LIN {X -0.292,Y -605.809,Z 406.567,A 0.000,B 0.000,C 90.000,E1 318.081} C_DIS
LIN {X 0.319,Y -611.269,Z 406.558,A 0.000,B 0.000,C 90.000,E1 316.458} C_DIS
LIN {X 0.160,Y -616.740,Z 406.550,A 0.000,B 0.000,C 90.000,E1 314.919} C_DIS
LIN {X -0.037,Y -623.235,Z 406.540,A 0.000,B 0.000,C 90.000,E1 313.137} C_DIS
LIN {X -0.138,Y -626.967,Z 406.534,A 0.000,B 0.000,C 90.000,E1 312.123} C_DIS
LIN {X -0.379,Y -632.521,Z 406.526,A 0.000,B 0.000,C 90.000,E1 310.620} C_DIS
LIN {X 0.008,Y -636.977,Z 406.518,A 0.000,B 0.000,C 90.000,E1 309.322} C_DIS
LIN {X 0.062,Y -641.986,Z 406.510,A 0.000,B 0.000,C 90.000,E1 307.810} C_DIS
LIN {X -0.197,Y -646.015,Z 406.503,A 0.000,B 0.000,C 90.000,E1 306.583} C_DIS
LIN {X 0.128,Y -649.848,Z 406.496,A 0.000,B 0.000,C 90.000,E1 305.311} C_DIS
LIN {X 0.149,Y -653.624,Z 406.489,A 0.000,B 0.000,C 90.000,E1 304.072} C_DIS
LIN {X -0.214,Y -657.959,Z 406.481,A 0.000,B 0.000,C 90.000,E1 302.625} C_DIS
LIN {X 0.054,Y -662.210,Z 406.473,A 0.000,B 0.000,C 90.000,E1 301.131} C_DIS
LIN {X 0.058,Y -666.331,Z 406.465,A 0.000,B 0.000,C 90.000,E1 299.667} C_DIS
LIN {X -0.349,Y -669.415,Z 406.458,A 0.000,B 0.000,C 90.000,E1 298.487} C_DIS
LIN {X 0.140,Y -671.219,Z 406.454,A 0.000,B 0.000,C 90.000,E1 297.719} C_DIS
LIN {X -0.141,Y -674.920,Z 406.445,A 0.000,B 0.000,C 90.000,E1 296.052} C_DIS
LIN {X -0.017,Y -676.898,Z 406.439,A 0.000,B 0.000,C 90.000,E1 295.079} C_DIS
LIN {X -0.164,Y -678.756,Z 406.434,A 0.000,B 0.000,C 90.000,E1 294.131} C_DIS
LIN {X 0.259,Y -680.450,Z 406.427,A 0.000,B 0.000,C 90.000,E1 292.898} C_DIS
LIN {X -0.046,Y -681.185,Z 406.423,A 0.000,B 0.000,C 90.000,E1 292.206} C_DIS
LIN {X 0.227,Y -681.792,Z 406.418,A 0.000,B 0.000,C 90.000,E1 291.227} C_DIS
LIN {X -0.127,Y -682.278,Z 406.413,A 0.000,B 0.000,C 90.000,E1 290.301} C_DIS
LIN {X -0.027,Y -682.414,Z 406.409,A 0.000,B 0.000,C 90.000,E1 289.577} C_DIS
LIN {X 0.259,Y -682.311,Z 406.404,A 0.000,B 0.000,C 90.000,E1 288.598} C_DIS
LIN {X 0.359,Y -681.967,Z 406.400,A 0.000,B 0.000,C 90.000,E1 287.873} C_DIS
LIN {X -0.234,Y -681.446,Z 406.394,A 0.000,B 0.000,C 90.000,E1 286.968} C_DIS
LIN {X 0.245,Y -680.502,Z 406.388,A 0.000,B 0.000,C 90.000,E1 285.733} C_DIS
LIN {X 0.357,Y -680.103,Z 406.385,A 0.000,B 0.000,C 90.000,E1 285.245} C_DIS
LIN {X 0.127,Y -678.512,Z 406.377,A 0.000,B 0.000,C 90.000,E1 283.828} C_DIS
LIN {X -0.041,Y -677.497,Z 406.372,A 0.000,B 0.000,C 90.000,E1 282.883} C_DIS
LIN {X -0.370,Y -676.465,Z 406.366,A 0.000,B 0.000,C 90.000,E1 281.951} C_DIS
LIN {X 0.335,Y -673.842,Z 406.354,A 0.000,B 0.000,C 90.000,E1 279.726} C_DIS
LIN {X -0.044,Y -671.489,Z 406.342,A 0.000,B 0.000,C 90.000,E1 277.587} C_DIS
LIN {X 0.176,Y -669.413,Z 406.330,A 0.000,B 0.000,C 90.000,E1 275.391} C_DIS
LIN {X -0.191,Y -667.809,Z 406.321,A 0.000,B 0.000,C 90.000,E1 273.726} C_DIS
LIN {X 0.028,Y -667.186,Z 406.317,A 0.000,B 0.000,C 90.000,E1 272.980} C_DIS
LIN {X 0.079,Y -665.517,Z 406.306,A 0.000,B 0.000,C 90.000,E1 271.031} C_DIS
LIN {X -0.082,Y -664.332,Z 406.299,A 0.000,B 0.000,C 90.000,E1 269.828} C_DIS
LIN {X 0.247,Y -663.720,Z 406.296,A 0.000,B 0.000,C 90.000,E1 269.312} C_DIS
LIN {X 0.078,Y -663.348,Z 406.295,A 0.000,B 0.000,C 90.000,E1 269.083} C_DIS
LIN {X -0.092,Y -663.132,Z 406.294,A 0.000,B 0.000,C 90.000,E1 268.854} C_DIS
LIN {X -0.278,Y -661.542,Z 406.287,A 0.000,B 0.000,C 90.000,E1 267.650} C_DIS
LIN {X 0.175,Y -659.739,Z 406.280,A 0.000,B 0.000,C 90.000,E1 266.388} C_DIS
LIN {X 0.316,Y -658.453,Z 406.276,A 0.000,B 0.000,C 90.000,E1 265.641} C_DIS
LIN {X -0.212,Y -656.934,Z 406.272,A 0.000,B 0.000,C 90.000,E1 264.951} C_DIS
LIN {X -0.239,Y -654.722,Z 406.266,A 0.000,B 0.000,C 90.000,E1 263.970} C_DIS
LIN {X 0.134,Y -651.558,Z 406.260,A 0.000,B 0.000,C 90.000,E1 262.704} C_DIS
LIN {X -0.260,Y -647.578,Z 406.251,A 0.000,B 0.000,C 90.000,E1 261.254} C_DIS
LIN {X 0.061,Y -643.908,Z 406.244,A 0.000,B 0.000,C 90.000,E1 259.982} C_DIS
LIN {X 0.256,Y -639.424,Z 406.236,A 0.000,B 0.000,C 90.000,E1 258.465} C_DIS
LIN {X -0.125,Y -634.791,Z 406.228,A 0.000,B 0.000,C 90.000,E1 256.992} C_DIS
LIN {X -0.219,Y -631.533,Z 406.222,A 0.000,B 0.000,C 90.000,E1 255.992} C_DIS
LIN {X 0.247,Y -628.136,Z 406.216,A 0.000,B 0.000,C 90.000,E1 254.936} C_DIS
LIN {X 0.009,Y -623.629,Z 406.209,A 0.000,B 0.000,C 90.000,E1 253.685} C_DIS
LIN {X -0.080,Y -619.921,Z 406.204,A 0.000,B 0.000,C 90.000,E1 252.670} C_DIS
LIN {X -0.030,Y -616.128,Z 406.198,A 0.000,B 0.000,C 90.000,E1 251.638} C_DIS
LIN {X -0.277,Y -611.249,Z 406.191,A 0.000,B 0.000,C 90.000,E1 250.369} C_DIS
LIN {X 0.167,Y -606.185,Z 406.184,A 0.000,B 0.000,C 90.000,E1 249.028} C_DIS
LIN {X 0.177,Y -600.901,Z 406.176,A 0.000,B 0.000,C 90.000,E1 247.720} C_DIS
LIN {X 0.192,Y -596.560,Z 406.171,A 0.000,B 0.000,C 90.000,E1 246.666} C_DIS
LIN {X -0.057,Y -589.938,Z 406.162,A 0.000,B 0.000,C 90.000,E1 245.101} C_DIS
LIN {X -0.316,Y -582.091,Z 406.151,A 0.000,B 0.000,C 90.000,E1 243.256} C_DIS
LIN {X -0.206,Y -576.508,Z 406.144,A 0.000,B 0.000,C 90.000,E1 241.897} C_DIS
LIN {X -0.254,Y -568.849,Z 406.133,A 0.000,B 0.000,C 90.000,E1 239.999} C_DIS
LIN {X -0.120,Y -560.426,Z 406.121,A 0.000,B 0.000,C 90.000,E1 237.788} C_DIS
LIN {X 0.063,Y -552.448,Z 406.109,A 0.000,B 0.000,C 90.000,E1 235.548} C_DIS
LIN {X 0.040,Y -547.623,Z 406.101,A 0.000,B 0.000,C 90.000,E1 234.149} C_DIS
LIN {X -0.181,Y -542.844,Z 406.093,A 0.000,B 0.000,C 90.000,E1 232.763} C_DIS
LIN {X -0.052,Y -538.005,Z 406.085,A 0.000,B 0.000,C 90.000,E1 231.331} C_DIS
LIN {X -0.102,Y -532.284,Z 406.076,A 0.000,B 0.000,C 90.000,E1 229.622} C_DIS
LIN {X -0.047,Y -525.042,Z 406.063,A 0.000,B 0.000,C 90.000,E1 227.310} C_DIS
LIN {X -0.064,Y -519.755,Z 406.053,A 0.000,B 0.000,C 90.000,E1 225.567} C_DIS
LIN {X 0.164,Y -514.572,Z 406.043,A 0.000,B 0.000,C 90.000,E1 223.785} C_DIS
LIN {X -0.087,Y -509.453,Z 406.034,A 0.000,B 0.000,C 90.000,E1 222.043} C_DIS
LIN {X 0.189,Y -503.698,Z 406.022,A 0.000,B 0.000,C 90.000,E1 219.930} C_DIS
LIN {X -0.009,Y -498.183,Z 406.010,A 0.000,B 0.000,C 90.000,E1 217.855} C_DIS
LIN {X -0.273,Y -494.353,Z 406.002,A 0.000,B 0.000,C 90.000,E1 216.377} C_DIS
LIN {X 0.179,Y -489.131,Z 405.990,A 0.000,B 0.000,C 90.000,E1 214.199} C_DIS
LIN {X 0.154,Y -485.555,Z 405.982,A 0.000,B 0.000,C 90.000,E1 212.673} C_DIS
LIN {X 0.011,Y -481.312,Z 405.971,A 0.000,B 0.000,C 90.000,E1 210.846} C_DIS
LIN {X -0.097,Y -476.330,Z 405.959,A 0.000,B 0.000,C 90.000,E1 208.693} C_DIS
LIN {X 0.003,Y -473.428,Z 405.952,A 0.000,B 0.000,C 90.000,E1 207.436} C_DIS
LIN {X 0.045,Y -470.495,Z 405.946,A 0.000,B 0.000,C 90.000,E1 206.181} C_DIS
LIN {X -0.225,Y -466.721,Z 405.937,A 0.000,B 0.000,C 90.000,E1 204.643} C_DIS
LIN {X 0.150,Y -463.676,Z 405.930,A 0.000,B 0.000,C 90.000,E1 203.334} C_DIS
LIN {X 0.237,Y -458.340,Z 405.917,A 0.000,B 0.000,C 90.000,E1 201.099} C_DIS
LIN {X 0.173,Y -452.612,Z 405.903,A 0.000,B 0.000,C 90.000,E1 198.544} C_DIS
LIN {X -0.081,Y -448.051,Z 405.891,A 0.000,B 0.000,C 90.000,E1 196.315} C_DIS
LIN {X -0.004,Y -443.326,Z 405.876,A 0.000,B 0.000,C 90.000,E1 193.703} C_DIS
LIN {X 0.182,Y -440.022,Z 405.865,A 0.000,B 0.000,C 90.000,E1 191.715} C_DIS
LIN {X -0.225,Y -435.417,Z 405.849,A 0.000,B 0.000,C 90.000,E1 188.803} C_DIS
LIN {X 0.182,Y -432.241,Z 405.836,A 0.000,B 0.000,C 90.000,E1 186.429} C_DIS
LIN {X -0.068,Y -429.477,Z 405.823,A 0.000,B 0.000,C 90.000,E1 184.131} C_DIS
LIN {X -0.109,Y -427.760,Z 405.814,A 0.000,B 0.000,C 90.000,E1 182.465} C_DIS
LIN {X 0.028,Y -425.302,Z 405.797,A 0.000,B 0.000,C 90.000,E1 179.427} C_DIS
LIN {X -0.092,Y -423.384,Z 405.773,A 0.000,B 0.000,C 90.000,E1 175.065} C_DIS
LIN {X -0.099,Y -423.234,Z 405.748,A 0.000,B 0.000,C 90.000,E1 170.679} C_DIS
LIN {X -0.112,Y -424.257,Z 405.731,A 0.000,B 0.000,C 90.000,E1 167.645} C_DIS
LIN {X 0.010,Y -425.939,Z 405.716,A 0.000,B 0.000,C 90.000,E1 164.936} C_DIS
LIN {X -0.203,Y -429.303,Z 405.696,A 0.000,B 0.000,C 90.000,E1 161.275} C_DIS
LIN {X 0.081,Y -432.036,Z 405.683,A 0.000,B 0.000,C 90.000,E1 158.901} C_DIS
LIN {X -0.211,Y -435.267,Z 405.670,A 0.000,B 0.000,C 90.000,E1 156.613} C_DIS
LIN {X 0.056,Y -441.290,Z 405.650,A 0.000,B 0.000,C 90.000,E1 152.948} C_DIS
LIN {X 0.241,Y -448.469,Z 405.630,A 0.000,B 0.000,C 90.000,E1 149.331} C_DIS
LIN {X -0.188,Y -453.751,Z 405.617,A 0.000,B 0.000,C 90.000,E1 147.120} C_DIS
LIN {X 0.011,Y -459.606,Z 405.605,A 0.000,B 0.000,C 90.000,E1 144.848} C_DIS
LIN {X 0.058,Y -467.981,Z 405.589,A 0.000,B 0.000,C 90.000,E1 141.984} C_DIS
LIN {X 0.168,Y -475.901,Z 405.575,A 0.000,B 0.000,C 90.000,E1 139.461} C_DIS
LIN {X -0.049,Y -479.829,Z 405.568,A 0.000,B 0.000,C 90.000,E1 138.243} C_DIS
LIN {X 0.117,Y -483.696,Z 405.561,A 0.000,B 0.000,C 90.000,E1 136.986} C_DIS
LIN {X 0.005,Y -487.291,Z 405.554,A 0.000,B 0.000,C 90.000,E1 135.769} C_DIS
LIN {X 0.117,Y -489.885,Z 405.549,A 0.000,B 0.000,C 90.000,E1 134.838} C_DIS
LIN {X 0.084,Y -492.873,Z 405.542,A 0.000,B 0.000,C 90.000,E1 133.623} C_DIS
LIN {X 0.271,Y -495.021,Z 405.537,A 0.000,B 0.000,C 90.000,E1 132.690} C_DIS
LIN {X -0.068,Y -496.262,Z 405.534,A 0.000,B 0.000,C 90.000,E1 132.123} C_DIS
LIN {X -0.032,Y -497.437,Z 405.531,A 0.000,B 0.000,C 90.000,E1 131.515} C_DIS
LIN {X -0.123,Y -498.910,Z 405.526,A 0.000,B 0.000,C 90.000,E1 130.620} C_DIS
LIN {X -0.003,Y -500.317,Z 405.519,A 0.000,B 0.000,C 90.000,E1 129.402} C_DIS
LIN {X -0.064,Y -500.918,Z 405.514,A 0.000,B 0.000,C 90.000,E1 128.508} C_DIS
LIN {X -0.032,Y -500.915,Z 405.509,A 0.000,B 0.000,C 90.000,E1 127.604} C_DIS
LIN {X 0.031,Y -500.539,Z 405.506,A 0.000,B 0.000,C 90.000,E1 126.996} C_DIS
LIN {X 0.068,Y -499.639,Z 405.501,A 0.000,B 0.000,C 90.000,E1 126.091} C_DIS
LIN {X -0.180,Y -498.858,Z 405.497,A 0.000,B 0.000,C 90.000,E1 125.518} C_DIS
LIN {X -0.156,Y -497.379,Z 405.492,A 0.000,B 0.000,C 90.000,E1 124.612} C_DIS
LIN {X 0.122,Y -496.834,Z 405.491,A 0.000,B 0.000,C 90.000,E1 124.278} C_DIS
LIN {X -0.021,Y -493.960,Z 405.484,A 0.000,B 0.000,C 90.000,E1 123.086} C_DIS
LIN {X 0.095,Y -492.235,Z 405.480,A 0.000,B 0.000,C 90.000,E1 122.467} C_DIS
LIN {X -0.064,Y -490.351,Z 405.477,A 0.000,B 0.000,C 90.000,E1 121.878} C_DIS
LIN {X 0.268,Y -487.154,Z 405.472,A 0.000,B 0.000,C 90.000,E1 120.924} C_DIS
LIN {X -0.159,Y -486.075,Z 405.470,A 0.000,B 0.000,C 90.000,E1 120.669} C_DIS
LIN {X -0.123,Y -482.428,Z 405.465,A 0.000,B 0.000,C 90.000,E1 119.745} C_DIS
LIN {X 0.064,Y -477.213,Z 405.458,A 0.000,B 0.000,C 90.000,E1 118.487} C_DIS
LIN {X -0.017,Y -473.070,Z 405.453,A 0.000,B 0.000,C 90.000,E1 117.564} C_DIS
LIN {X -0.180,Y -467.971,Z 405.447,A 0.000,B 0.000,C 90.000,E1 116.488} C_DIS
LIN {X 0.066,Y -459.764,Z 405.437,A 0.000,B 0.000,C 90.000,E1 114.719} C_DIS
LIN {X -0.135,Y -450.626,Z 405.427,A 0.000,B 0.000,C 90.000,E1 112.823} C_DIS
LIN {X -0.023,Y -449.846,Z 405.426,A 0.000,B 0.000,C 90.000,E1 112.642} C_DIS
LIN {X -0.063,Y -449.857,Z 405.426,A 0.000,B 0.000,C 90.000,E1 112.642} C_DIS
LIN {X 0.142,Y -456.999,Z 405.411,A 0.000,B 0.000,C 90.000,E1 109.885} C_DIS
LIN {X -0.050,Y -458.255,Z 405.407,A 0.000,B 0.000,C 90.000,E1 109.268} C_DIS
LIN {X 0.148,Y -466.417,Z 405.386,A 0.000,B 0.000,C 90.000,E1 105.426} C_DIS
LIN {X -0.129,Y -467.925,Z 405.382,A 0.000,B 0.000,C 90.000,E1 104.828} C_DIS
LIN {X -0.015,Y -475.501,Z 405.358,A 0.000,B 0.000,C 90.000,E1 100.423} C_DIS
LIN {X -0.263,Y -476.141,Z 405.356,A 0.000,B 0.000,C 90.000,E1 100.141} C_DIS
LIN {X 0.020,Y -482.054,Z 405.330,A 0.000,B 0.000,C 90.000,E1 95.454} C_DIS
LIN {X -0.190,Y -485.484,Z 405.305,A 0.000,B 0.000,C 90.000,E1 90.859} C_DIS
LIN {X -0.157,Y -486.386,Z 405.281,A 0.000,B 0.000,C 90.000,E1 86.560} C_DIS
LIN {X 0.153,Y -486.363,Z 405.279,A 0.000,B 0.000,C 90.000,E1 86.216} C_DIS
LIN {X 0.236,Y -484.689,Z 405.254,A 0.000,B 0.000,C 90.000,E1 81.602} C_DIS
LIN {X -0.016,Y -483.031,Z 405.245,A 0.000,B 0.000,C 90.000,E1 80.095} C_DIS
LIN {X 0.135,Y -480.621,Z 405.228,A 0.000,B 0.000,C 90.000,E1 76.992} C_DIS
LIN {X -0.007,Y -480.289,Z 405.226,A 0.000,B 0.000,C 90.000,E1 76.700} C_DIS
LIN {X -0.103,Y -474.111,Z 405.200,A 0.000,B 0.000,C 90.000,E1 72.054} C_DIS
LIN {X -0.058,Y -469.651,Z 405.187,A 0.000,B 0.000,C 90.000,E1 69.699} C_DIS
LIN {X -0.099,Y -469.650,Z 405.187,A 0.000,B 0.000,C 90.000,E1 69.699} C_DIS
LIN {X -0.162,Y -479.044,Z 405.180,A 0.000,B 0.000,C 90.000,E1 68.465} C_DIS
LIN {X 0.046,Y -487.179,Z 405.174,A 0.000,B 0.000,C 90.000,E1 67.358} C_DIS
LIN {X 0.117,Y -494.115,Z 405.169,A 0.000,B 0.000,C 90.000,E1 66.433} C_DIS
LIN {X 0.013,Y -500.651,Z 405.164,A 0.000,B 0.000,C 90.000,E1 65.537} C_DIS
LIN {X -0.038,Y -505.900,Z 405.160,A 0.000,B 0.000,C 90.000,E1 64.793} C_DIS
LIN {X -0.007,Y -511.657,Z 405.155,A 0.000,B 0.000,C 90.000,E1 63.896} C_DIS
LIN {X 0.262,Y -516.102,Z 405.151,A 0.000,B 0.000,C 90.000,E1 63.127} C_DIS
LIN {X 0.116,Y -520.139,Z 405.147,A 0.000,B 0.000,C 90.000,E1 62.410} C_DIS
LIN {X 0.083,Y -522.373,Z 405.144,A 0.000,B 0.000,C 90.000,E1 61.975} C_DIS
LIN {X -0.010,Y -525.740,Z 405.140,A 0.000,B 0.000,C 90.000,E1 61.257} C_DIS
LIN {X -0.075,Y -528.710,Z 405.136,A 0.000,B 0.000,C 90.000,E1 60.539} C_DIS
LIN {X -0.005,Y -531.910,Z 405.132,A 0.000,B 0.000,C 90.000,E1 59.665} C_DIS
LIN {X -0.305,Y -532.888,Z 405.130,A 0.000,B 0.000,C 90.000,E1 59.410} C_DIS
LIN {X -0.186,Y -535.279,Z 405.125,A 0.000,B 0.000,C 90.000,E1 58.535} C_DIS
LIN {X -0.033,Y -536.723,Z 405.122,A 0.000,B 0.000,C 90.000,E1 57.946} C_DIS
LIN {X -0.035,Y -538.263,Z 405.117,A 0.000,B 0.000,C 90.000,E1 57.089} C_DIS
LIN {X 0.136,Y -539.104,Z 405.114,A 0.000,B 0.000,C 90.000,E1 56.501} C_DIS
LIN {X -0.128,Y -539.955,Z 405.109,A 0.000,B 0.000,C 90.000,E1 55.674} C_DIS
LIN {X -0.075,Y -540.394,Z 405.105,A 0.000,B 0.000,C 90.000,E1 54.815} C_DIS
LIN {X -0.328,Y -540.511,Z 405.100,A 0.000,B 0.000,C 90.000,E1 53.989} C_DIS
LIN {X -0.265,Y -540.225,Z 405.095,A 0.000,B 0.000,C 90.000,E1 53.130} C_DIS
LIN {X -0.204,Y -539.735,Z 405.090,A 0.000,B 0.000,C 90.000,E1 52.271} C_DIS
LIN {X 0.199,Y -538.721,Z 405.084,A 0.000,B 0.000,C 90.000,E1 51.090} C_DIS
LIN {X -0.178,Y -537.800,Z 405.079,A 0.000,B 0.000,C 90.000,E1 50.275} C_DIS
LIN {X 0.192,Y -536.392,Z 405.073,A 0.000,B 0.000,C 90.000,E1 49.094} C_DIS
LIN {X 0.071,Y -533.908,Z 405.063,A 0.000,B 0.000,C 90.000,E1 47.391} C_DIS
LIN {X -0.151,Y -530.898,Z 405.052,A 0.000,B 0.000,C 90.000,E1 45.405} C_DIS
LIN {X -0.021,Y -528.478,Z 405.043,A 0.000,B 0.000,C 90.000,E1 43.662} C_DIS
LIN {X 0.094,Y -526.657,Z 405.035,A 0.000,B 0.000,C 90.000,E1 42.204} C_DIS
LIN {X 0.159,Y -524.464,Z 405.025,A 0.000,B 0.000,C 90.000,E1 40.458} C_DIS
LIN {X -0.118,Y -522.730,Z 405.017,A 0.000,B 0.000,C 90.000,E1 39.036} C_DIS
LIN {X -0.024,Y -520.969,Z 405.009,A 0.000,B 0.000,C 90.000,E1 37.569} C_DIS
LIN {X 0.083,Y -518.720,Z 404.999,A 0.000,B 0.000,C 90.000,E1 35.804} C_DIS
LIN {X 0.207,Y -516.855,Z 404.991,A 0.000,B 0.000,C 90.000,E1 34.326} C_DIS
LIN {X -0.074,Y -514.486,Z 404.981,A 0.000,B 0.000,C 90.000,E1 32.594} C_DIS
LIN {X 0.183,Y -512.099,Z 404.971,A 0.000,B 0.000,C 90.000,E1 30.797} C_DIS
LIN {X 0.030,Y -509.398,Z 404.960,A 0.000,B 0.000,C 90.000,E1 28.743} C_DIS
LIN {X 0.091,Y -506.540,Z 404.947,A 0.000,B 0.000,C 90.000,E1 26.360} C_DIS
LIN {X 0.217,Y -504.245,Z 404.935,A 0.000,B 0.000,C 90.000,E1 24.259} C_DIS
LIN {X -0.054,Y -501.964,Z 404.922,A 0.000,B 0.000,C 90.000,E1 21.897} C_DIS
LIN {X -0.209,Y -499.869,Z 404.907,A 0.000,B 0.000,C 90.000,E1 19.214} C_DIS
LIN {X -0.141,Y -498.656,Z 404.897,A 0.000,B 0.000,C 90.000,E1 17.402} C_DIS
LIN {X -0.251,Y -497.468,Z 404.887,A 0.000,B 0.000,C 90.000,E1 15.607} C_DIS
LIN {X -0.014,Y -496.319,Z 404.875,A 0.000,B 0.000,C 90.000,E1 13.467} C_DIS
LIN {X 0.073,Y -495.186,Z 404.858,A 0.000,B 0.000,C 90.000,E1 10.433} C_DIS
LIN {X -0.120,Y -494.821,Z 404.840,A 0.000,B 0.000,C 90.000,E1 7.125} C_DIS
LIN {X 0.234,Y -495.290,Z 404.824,A 0.000,B 0.000,C 90.000,E1 4.359} C_DIS
LIN {X 0.114,Y -497.276,Z 404.804,A 0.000,B 0.000,C 90.000,E1 0.745} C_DIS
LIN {X 0.050,Y -500.917,Z 404.784,A 0.000,B 0.000,C 90.000,E1 357.078} C_DIS
LIN {X 0.097,Y -504.640,Z 404.769,A 0.000,B 0.000,C 90.000,E1 354.375} C_DIS
LIN {X 0.231,Y -510.046,Z 404.751,A 0.000,B 0.000,C 90.000,E1 351.084} C_DIS
LIN {X -0.206,Y -517.264,Z 404.731,A 0.000,B 0.000,C 90.000,E1 347.589} C_DIS
LIN {X -0.020,Y -523.695,Z 404.716,A 0.000,B 0.000,C 90.000,E1 344.936} C_DIS
LIN {X 0.138,Y -529.654,Z 404.703,A 0.000,B 0.000,C 90.000,E1 342.598} C_DIS
LIN {X -0.256,Y -534.266,Z 404.694,A 0.000,B 0.000,C 90.000,E1 340.913} C_DIS
LIN {X -0.166,Y -539.823,Z 404.683,A 0.000,B 0.000,C 90.000,E1 338.901} C_DIS
LIN {X 0.015,Y -544.710,Z 404.673,A 0.000,B 0.000,C 90.000,E1 337.177} C_DIS
LIN {X 0.012,Y -549.662,Z 404.664,A 0.000,B 0.000,C 90.000,E1 335.485} C_DIS
LIN {X -0.146,Y -554.736,Z 404.655,A 0.000,B 0.000,C 90.000,E1 333.819} C_DIS
LIN {X 0.099,Y -560.909,Z 404.644,A 0.000,B 0.000,C 90.000,E1 331.847} C_DIS
LIN {X 0.056,Y -564.471,Z 404.638,A 0.000,B 0.000,C 90.000,E1 330.745} C_DIS
LIN {X -0.335,Y -569.001,Z 404.630,A 0.000,B 0.000,C 90.000,E1 329.410} C_DIS
LIN {X 0.142,Y -573.488,Z 404.622,A 0.000,B 0.000,C 90.000,E1 327.995} C_DIS
LIN {X 0.053,Y -578.802,Z 404.613,A 0.000,B 0.000,C 90.000,E1 326.373} C_DIS
LIN {X 0.088,Y -585.073,Z 404.603,A 0.000,B 0.000,C 90.000,E1 324.482} C_DIS
LIN {X -0.199,Y -591.451,Z 404.592,A 0.000,B 0.000,C 90.000,E1 322.637} C_DIS
LIN {X -0.219,Y -598.891,Z 404.581,A 0.000,B 0.000,C 90.000,E1 320.517} C_DIS
LIN {X -0.190,Y -602.702,Z 404.575,A 0.000,B 0.000,C 90.000,E1 319.461} C_DIS
LIN {X -0.307,Y -607.397,Z 404.567,A 0.000,B 0.000,C 90.000,E1 318.162} C_DIS
LIN {X 0.068,Y -611.968,Z 404.560,A 0.000,B 0.000,C 90.000,E1 316.824} C_DIS
LIN {X -0.343,Y -616.514,Z 404.553,A 0.000,B 0.000,C 90.000,E1 315.567} C_DIS
LIN {X 0.192,Y -623.936,Z 404.542,A 0.000,B 0.000,C 90.000,E1 313.461} C_DIS
LIN {X 0.312,Y -629.479,Z 404.533,A 0.000,B 0.000,C 90.000,E1 311.919} C_DIS
LIN {X -0.233,Y -634.141,Z 404.526,A 0.000,B 0.000,C 90.000,E1 310.701} C_DIS
LIN {X 0.185,Y -638.585,Z 404.519,A 0.000,B 0.000,C 90.000,E1 309.402} C_DIS
LIN {X -0.134,Y -642.816,Z 404.512,A 0.000,B 0.000,C 90.000,E1 308.177} C_DIS
LIN {X 0.011,Y -646.880,Z 404.505,A 0.000,B 0.000,C 90.000,E1 306.916} C_DIS
LIN {X -0.126,Y -651.561,Z 404.497,A 0.000,B 0.000,C 90.000,E1 305.438} C_DIS
LIN {X 0.371,Y -655.990,Z 404.489,A 0.000,B 0.000,C 90.000,E1 303.913} C_DIS
LIN {X 0.026,Y -658.914,Z 404.483,A 0.000,B 0.000,C 90.000,E1 302.959} C_DIS
LIN {X -0.281,Y -661.770,Z 404.478,A 0.000,B 0.000,C 90.000,E1 302.005} C_DIS
LIN {X -0.286,Y -665.988,Z 404.470,A 0.000,B 0.000,C 90.000,E1 300.541} C_DIS
LIN {X 0.063,Y -668.735,Z 404.464,A 0.000,B 0.000,C 90.000,E1 299.539} C_DIS
LIN {X 0.119,Y -671.176,Z 404.459,A 0.000,B 0.000,C 90.000,E1 298.565} C_DIS
LIN {X 0.209,Y -673.459,Z 404.453,A 0.000,B 0.000,C 90.000,E1 297.590} C_DIS
LIN {X 0.090,Y -676.595,Z 404.445,A 0.000,B 0.000,C 90.000,E1 296.155} C_DIS
LIN {X -0.252,Y -678.133,Z 404.441,A 0.000,B 0.000,C 90.000,E1 295.463} C_DIS
LIN {X 0.238,Y -679.925,Z 404.436,A 0.000,B 0.000,C 90.000,E1 294.463} C_DIS
LIN {X 0.132,Y -681.298,Z 404.431,A 0.000,B 0.000,C 90.000,E1 293.515} C_DIS
LIN {X -0.164,Y -682.122,Z 404.427,A 0.000,B 0.000,C 90.000,E1 292.823} C_DIS
LIN {X -0.027,Y -682.523,Z 404.424,A 0.000,B 0.000,C 90.000,E1 292.333} C_DIS
LIN {X 0.316,Y -682.912,Z 404.420,A 0.000,B 0.000,C 90.000,E1 291.589} C_DIS
LIN {X -0.072,Y -683.284,Z 404.414,A 0.000,B 0.000,C 90.000,E1 290.429} C_DIS
LIN {X 0.080,Y -683.327,Z 404.411,A 0.000,B 0.000,C 90.000,E1 289.939} C_DIS
LIN {X 0.341,Y -683.100,Z 404.404,A 0.000,B 0.000,C 90.000,E1 288.725} C_DIS
LIN {X -0.232,Y -682.613,Z 404.399,A 0.000,B 0.000,C 90.000,E1 287.819} C_DIS
LIN {X -0.128,Y -682.226,Z 404.395,A 0.000,B 0.000,C 90.000,E1 287.094} C_DIS
LIN {X -0.102,Y -681.144,Z 404.388,A 0.000,B 0.000,C 90.000,E1 285.898} C_DIS
LIN {X -0.171,Y -680.632,Z 404.386,A 0.000,B 0.000,C 90.000,E1 285.426} C_DIS
LIN {X -0.385,Y -678.739,Z 404.378,A 0.000,B 0.000,C 90.000,E1 284.008} C_DIS
LIN {X 0.113,Y -677.597,Z 404.372,A 0.000,B 0.000,C 90.000,E1 283.008} C_DIS
LIN {X -0.069,Y -676.406,Z 404.367,A 0.000,B 0.000,C 90.000,E1 282.063} C_DIS
LIN {X -0.156,Y -673.613,Z 404.355,A 0.000,B 0.000,C 90.000,E1 279.905} C_DIS
LIN {X 0.058,Y -670.894,Z 404.342,A 0.000,B 0.000,C 90.000,E1 277.473} C_DIS
LIN {X -0.299,Y -669.073,Z 404.331,A 0.000,B 0.000,C 90.000,E1 275.568} C_DIS
LIN {X 0.170,Y -667.833,Z 404.323,A 0.000,B 0.000,C 90.000,E1 274.073} C_DIS
LIN {X 0.283,Y -666.289,Z 404.312,A 0.000,B 0.000,C 90.000,E1 272.121} C_DIS
LIN {X 0.152,Y -665.532,Z 404.305,A 0.000,B 0.000,C 90.000,E1 270.917} C_DIS
LIN {X -0.009,Y -664.468,Z 404.298,A 0.000,B 0.000,C 90.000,E1 269.714} C_DIS
LIN {X -0.188,Y -663.195,Z 404.292,A 0.000,B 0.000,C 90.000,E1 268.511} C_DIS
LIN {X -0.022,Y -662.406,Z 404.288,A 0.000,B 0.000,C 90.000,E1 267.764} C_DIS
LIN {X -0.213,Y -660.652,Z 404.281,A 0.000,B 0.000,C 90.000,E1 266.560} C_DIS
LIN {X -0.061,Y -659.439,Z 404.277,A 0.000,B 0.000,C 90.000,E1 265.812} C_DIS
LIN {X 0.078,Y -658.037,Z 404.273,A 0.000,B 0.000,C 90.000,E1 265.065} C_DIS
LIN {X -0.138,Y -655.412,Z 404.266,A 0.000,B 0.000,C 90.000,E1 263.856} C_DIS
LIN {X -0.184,Y -653.004,Z 404.260,A 0.000,B 0.000,C 90.000,E1 262.875} C_DIS
LIN {X 0.240,Y -649.847,Z 404.254,A 0.000,B 0.000,C 90.000,E1 261.602} C_DIS
LIN {X -0.282,Y -647.850,Z 404.249,A 0.000,B 0.000,C 90.000,E1 260.905} C_DIS
LIN {X 0.041,Y -644.246,Z 404.242,A 0.000,B 0.000,C 90.000,E1 259.634} C_DIS
LIN {X 0.241,Y -639.806,Z 404.234,A 0.000,B 0.000,C 90.000,E1 258.117} C_DIS
LIN {X -0.137,Y -635.149,Z 404.226,A 0.000,B 0.000,C 90.000,E1 256.645} C_DIS
LIN {X -0.230,Y -631.883,Z 404.220,A 0.000,B 0.000,C 90.000,E1 255.644} C_DIS
LIN {X -0.017,Y -629.350,Z 404.216,A 0.000,B 0.000,C 90.000,E1 254.866} C_DIS
LIN {X -0.224,Y -624.838,Z 404.209,A 0.000,B 0.000,C 90.000,E1 253.614} C_DIS
LIN {X 0.083,Y -620.185,Z 404.202,A 0.000,B 0.000,C 90.000,E1 252.308} C_DIS
LIN {X -0.101,Y -615.381,Z 404.195,A 0.000,B 0.000,C 90.000,E1 251.040} C_DIS
LIN {X -0.158,Y -610.427,Z 404.187,A 0.000,B 0.000,C 90.000,E1 249.752} C_DIS
LIN {X -0.232,Y -606.311,Z 404.182,A 0.000,B 0.000,C 90.000,E1 248.720} C_DIS
LIN {X -0.213,Y -600.977,Z 404.174,A 0.000,B 0.000,C 90.000,E1 247.411} C_DIS
LIN {X -0.197,Y -596.584,Z 404.169,A 0.000,B 0.000,C 90.000,E1 246.357} C_DIS
LIN {X -0.096,Y -591.052,Z 404.161,A 0.000,B 0.000,C 90.000,E1 245.025} C_DIS
LIN {X 0.321,Y -584.328,Z 404.152,A 0.000,B 0.000,C 90.000,E1 243.384} C_DIS
LIN {X 0.325,Y -577.641,Z 404.143,A 0.000,B 0.000,C 90.000,E1 241.769} C_DIS
LIN {X -0.316,Y -571.065,Z 404.134,A 0.000,B 0.000,C 90.000,E1 240.205} C_DIS
LIN {X -0.025,Y -561.599,Z 404.121,A 0.000,B 0.000,C 90.000,E1 237.709} C_DIS
LIN {X 0.265,Y -552.679,Z 404.107,A 0.000,B 0.000,C 90.000,E1 235.182} C_DIS
LIN {X -0.192,Y -547.889,Z 404.099,A 0.000,B 0.000,C 90.000,E1 233.829} C_DIS
LIN {X 0.036,Y -543.124,Z 404.091,A 0.000,B 0.000,C 90.000,E1 232.396} C_DIS
LIN {X -0.234,Y -537.353,Z 404.082,A 0.000,B 0.000,C 90.000,E1 230.723} C_DIS
LIN {X -0.294,Y -531.639,Z 404.072,A 0.000,B 0.000,C 90.000,E1 229.013} C_DIS
LIN {X -0.209,Y -525.396,Z 404.061,A 0.000,B 0.000,C 90.000,E1 226.986} C_DIS
LIN {X 0.226,Y -521.008,Z 404.053,A 0.000,B 0.000,C 90.000,E1 225.486} C_DIS
LIN {X -0.251,Y -515.788,Z 404.043,A 0.000,B 0.000,C 90.000,E1 223.785} C_DIS
LIN {X 0.156,Y -509.829,Z 404.032,A 0.000,B 0.000,C 90.000,E1 221.676} C_DIS
LIN {X -0.267,Y -504.104,Z 404.020,A 0.000,B 0.000,C 90.000,E1 219.644} C_DIS
LIN {X -0.050,Y -498.614,Z 404.008,A 0.000,B 0.000,C 90.000,E1 217.523} C_DIS
LIN {X -0.006,Y -494.773,Z 404.000,A 0.000,B 0.000,C 90.000,E1 216.011} C_DIS
LIN {X -0.075,Y -490.323,Z 403.990,A 0.000,B 0.000,C 90.000,E1 214.199} C_DIS
LIN {X 0.094,Y -487.460,Z 403.983,A 0.000,B 0.000,C 90.000,E1 212.959} C_DIS
LIN {X 0.224,Y -482.503,Z 403.971,A 0.000,B 0.000,C 90.000,E1 210.797} C_DIS
LIN {X 0.183,Y -478.240,Z 403.961,A 0.000,B 0.000,C 90.000,E1 208.949} C_DIS
LIN {X 0.276,Y -474.626,Z 403.952,A 0.000,B 0.000,C 90.000,E1 207.385} C_DIS
LIN {X -0.085,Y -471.708,Z 403.945,A 0.000,B 0.000,C 90.000,E1 206.181} C_DIS
LIN {X 0.094,Y -467.916,Z 403.937,A 0.000,B 0.000,C 90.000,E1 204.591} C_DIS
LIN {X 0.004,Y -464.067,Z 403.928,A 0.000,B 0.000,C 90.000,E1 203.025} C_DIS
LIN {X 0.102,Y -458.789,Z 403.916,A 0.000,B 0.000,C 90.000,E1 200.791} C_DIS
LIN {X 0.157,Y -453.803,Z 403.903,A 0.000,B 0.000,C 90.000,E1 198.544} C_DIS
LIN {X -0.066,Y -449.211,Z 403.891,A 0.000,B 0.000,C 90.000,E1 196.315} C_DIS
LIN {X 0.046,Y -444.445,Z 403.876,A 0.000,B 0.000,C 90.000,E1 193.703} C_DIS
LIN {X -0.173,Y -441.125,Z 403.865,A 0.000,B 0.000,C 90.000,E1 191.771} C_DIS
LIN {X -0.112,Y -436.498,Z 403.849,A 0.000,B 0.000,C 90.000,E1 188.803} C_DIS
LIN {X 0.201,Y -433.715,Z 403.838,A 0.000,B 0.000,C 90.000,E1 186.777} C_DIS
LIN {X 0.101,Y -430.491,Z 403.823,A 0.000,B 0.000,C 90.000,E1 184.131} C_DIS
LIN {X -0.130,Y -427.823,Z 403.808,A 0.000,B 0.000,C 90.000,E1 181.489} C_DIS
LIN {X 0.179,Y -425.118,Z 403.786,A 0.000,B 0.000,C 90.000,E1 177.421} C_DIS
LIN {X -0.122,Y -424.182,Z 403.769,A 0.000,B 0.000,C 90.000,E1 174.432} C_DIS
LIN {X -0.029,Y -424.234,Z 403.745,A 0.000,B 0.000,C 90.000,E1 170.038} C_DIS
LIN {X 0.088,Y -425.495,Z 403.728,A 0.000,B 0.000,C 90.000,E1 166.992} C_DIS
LIN {X 0.117,Y -428.470,Z 403.705,A 0.000,B 0.000,C 90.000,E1 162.960} C_DIS
LIN {X 0.121,Y -431.682,Z 403.689,A 0.000,B 0.000,C 90.000,E1 159.953} C_DIS
LIN {X 0.038,Y -435.159,Z 403.674,A 0.000,B 0.000,C 90.000,E1 157.305} C_DIS
LIN {X 0.038,Y -439.749,Z 403.657,A 0.000,B 0.000,C 90.000,E1 154.332} C_DIS
LIN {X 0.064,Y -443.334,Z 403.647,A 0.000,B 0.000,C 90.000,E1 152.359} C_DIS
LIN {X -0.121,Y -450.072,Z 403.628,A 0.000,B 0.000,C 90.000,E1 149.125} C_DIS
LIN {X 0.220,Y -456.258,Z 403.614,A 0.000,B 0.000,C 90.000,E1 146.501} C_DIS
LIN {X -0.138,Y -463.270,Z 403.600,A 0.000,B 0.000,C 90.000,E1 143.989} C_DIS
LIN {X 0.127,Y -469.952,Z 403.588,A 0.000,B 0.000,C 90.000,E1 141.743} C_DIS
LIN {X 0.210,Y -476.948,Z 403.575,A 0.000,B 0.000,C 90.000,E1 139.542} C_DIS
LIN {X 0.129,Y -481.950,Z 403.567,A 0.000,B 0.000,C 90.000,E1 138.000} C_DIS
LIN {X -0.002,Y -485.756,Z 403.560,A 0.000,B 0.000,C 90.000,E1 136.782} C_DIS
LIN {X 0.059,Y -490.238,Z 403.551,A 0.000,B 0.000,C 90.000,E1 135.243} C_DIS
LIN {X -0.139,Y -492.644,Z 403.546,A 0.000,B 0.000,C 90.000,E1 134.352} C_DIS
LIN {X -0.135,Y -495.607,Z 403.540,A 0.000,B 0.000,C 90.000,E1 133.137} C_DIS
LIN {X -0.106,Y -496.965,Z 403.536,A 0.000,B 0.000,C 90.000,E1 132.528} C_DIS
LIN {X 0.128,Y -498.766,Z 403.531,A 0.000,B 0.000,C 90.000,E1 131.595} C_DIS
LIN {X -0.076,Y -500.703,Z 403.525,A 0.000,B 0.000,C 90.000,E1 130.415} C_DIS
LIN {X 0.196,Y -501.756,Z 403.520,A 0.000,B 0.000,C 90.000,E1 129.483} C_DIS
LIN {X -0.044,Y -502.259,Z 403.516,A 0.000,B 0.000,C 90.000,E1 128.910} C_DIS
LIN {X 0.036,Y -502.590,Z 403.513,A 0.000,B 0.000,C 90.000,E1 128.302} C_DIS
LIN {X 0.090,Y -502.513,Z 403.508,A 0.000,B 0.000,C 90.000,E1 127.397} C_DIS
LIN {X 0.050,Y -501.822,Z 403.503,A 0.000,B 0.000,C 90.000,E1 126.503} C_DIS
LIN {X 0.103,Y -500.791,Z 403.498,A 0.000,B 0.000,C 90.000,E1 125.598} C_DIS
LIN {X 0.149,Y -499.355,Z 403.493,A 0.000,B 0.000,C 90.000,E1 124.692} C_DIS
LIN {X -0.104,Y -498.269,Z 403.490,A 0.000,B 0.000,C 90.000,E1 124.119} C_DIS
LIN {X -0.090,Y -496.084,Z 403.484,A 0.000,B 0.000,C 90.000,E1 123.214} C_DIS
LIN {X -0.226,Y -494.443,Z 403.481,A 0.000,B 0.000,C 90.000,E1 122.625} C_DIS
LIN {X -0.104,Y -492.607,Z 403.478,A 0.000,B 0.000,C 90.000,E1 122.005} C_DIS
LIN {X 0.001,Y -489.483,Z 403.473,A 0.000,B 0.000,C 90.000,E1 121.082} C_DIS
LIN {X 0.079,Y -487.267,Z 403.469,A 0.000,B 0.000,C 90.000,E1 120.463} C_DIS
LIN {X 0.125,Y -483.561,Z 403.464,A 0.000,B 0.000,C 90.000,E1 119.539} C_DIS
LIN {X -0.102,Y -479.041,Z 403.458,A 0.000,B 0.000,C 90.000,E1 118.487} C_DIS
LIN {X -0.199,Y -473.425,Z 403.451,A 0.000,B 0.000,C 90.000,E1 117.257} C_DIS
LIN {X -0.198,Y -466.742,Z 403.444,A 0.000,B 0.000,C 90.000,E1 115.848} C_DIS
LIN {X 0.099,Y -459.960,Z 403.436,A 0.000,B 0.000,C 90.000,E1 114.387} C_DIS
LIN {X -0.177,Y -452.289,Z 403.427,A 0.000,B 0.000,C 90.000,E1 112.823} C_DIS
LIN {X -0.005,Y -450.414,Z 403.425,A 0.000,B 0.000,C 90.000,E1 112.408} C_DIS
LIN {X 0.127,Y -450.412,Z 403.424,A 0.000,B 0.000,C 90.000,E1 112.386} C_DIS
LIN {X -0.151,Y -457.399,Z 403.410,A 0.000,B 0.000,C 90.000,E1 109.758} C_DIS
LIN {X -0.067,Y -466.040,Z 403.387,A 0.000,B 0.000,C 90.000,E1 105.607} C_DIS
LIN {X 0.107,Y -467.608,Z 403.383,A 0.000,B 0.000,C 90.000,E1 104.954} C_DIS
LIN {X 0.105,Y -469.065,Z 403.378,A 0.000,B 0.000,C 90.000,E1 104.008} C_DIS
LIN {X 0.065,Y -475.834,Z 403.357,A 0.000,B 0.000,C 90.000,E1 100.254} C_DIS
LIN {X -0.096,Y -476.319,Z 403.355,A 0.000,B 0.000,C 90.000,E1 99.962} C_DIS
LIN {X -0.149,Y -481.813,Z 403.331,A 0.000,B 0.000,C 90.000,E1 95.625} C_DIS
LIN {X 0.177,Y -482.177,Z 403.329,A 0.000,B 0.000,C 90.000,E1 95.277} C_DIS
LIN {X 0.112,Y -485.324,Z 403.306,A 0.000,B 0.000,C 90.000,E1 90.974} C_DIS
LIN {X -0.064,Y -485.535,Z 403.304,A 0.000,B 0.000,C 90.000,E1 90.688} C_DIS
LIN {X 0.144,Y -486.327,Z 403.282,A 0.000,B 0.000,C 90.000,E1 86.674} C_DIS
LIN {X -0.207,Y -486.294,Z 403.278,A 0.000,B 0.000,C 90.000,E1 86.102} C_DIS
LIN {X -0.003,Y -484.695,Z 403.254,A 0.000,B 0.000,C 90.000,E1 81.781} C_DIS
LIN {X -0.134,Y -484.581,Z 403.253,A 0.000,B 0.000,C 90.000,E1 81.489} C_DIS
LIN {X -0.254,Y -480.518,Z 403.227,A 0.000,B 0.000,C 90.000,E1 76.881} C_DIS
LIN {X 0.110,Y -474.270,Z 403.201,A 0.000,B 0.000,C 90.000,E1 72.181} C_DIS
LIN {X 0.078,Y -473.815,Z 403.199,A 0.000,B 0.000,C 90.000,E1 71.873} C_DIS
LIN {X 0.196,Y -470.020,Z 403.188,A 0.000,B 0.000,C 90.000,E1 69.880} C_DIS
LIN {X 0.156,Y -470.045,Z 403.188,A 0.000,B 0.000,C 90.000,E1 69.880} C_DIS
LIN {X -0.153,Y -478.687,Z 403.182,A 0.000,B 0.000,C 90.000,E1 68.773} C_DIS
LIN {X -0.167,Y -487.876,Z 403.175,A 0.000,B 0.000,C 90.000,E1 67.539} C_DIS
LIN {X -0.065,Y -494.799,Z 403.170,A 0.000,B 0.000,C 90.000,E1 66.613} C_DIS
LIN {X 0.036,Y -500.239,Z 403.166,A 0.000,B 0.000,C 90.000,E1 65.845} C_DIS
LIN {X -0.206,Y -506.540,Z 403.161,A 0.000,B 0.000,C 90.000,E1 64.973} C_DIS
LIN {X 0.115,Y -513.114,Z 403.155,A 0.000,B 0.000,C 90.000,E1 63.896} C_DIS
LIN {X -0.061,Y -517.467,Z 403.151,A 0.000,B 0.000,C 90.000,E1 63.179} C_DIS
LIN {X 0.025,Y -521.450,Z 403.147,A 0.000,B 0.000,C 90.000,E1 62.436} C_DIS
LIN {X 0.080,Y -524.228,Z 403.144,A 0.000,B 0.000,C 90.000,E1 61.847} C_DIS
LIN {X -0.146,Y -526.267,Z 403.141,A 0.000,B 0.000,C 90.000,E1 61.435} C_DIS
LIN {X -0.205,Y -529.189,Z 403.137,A 0.000,B 0.000,C 90.000,E1 60.717} C_DIS
LIN {X -0.088,Y -531.341,Z 403.134,A 0.000,B 0.000,C 90.000,E1 60.127} C_DIS
LIN {X 0.039,Y -533.279,Z 403.131,A 0.000,B 0.000,C 90.000,E1 59.537} C_DIS
LIN {X 0.166,Y -535.733,Z 403.126,A 0.000,B 0.000,C 90.000,E1 58.663} C_DIS
LIN {X -0.131,Y -537.168,Z 403.123,A 0.000,B 0.000,C 90.000,E1 58.122} C_DIS
LIN {X 0.038,Y -538.856,Z 403.118,A 0.000,B 0.000,C 90.000,E1 57.248} C_DIS
LIN {X -0.228,Y -540.087,Z 403.113,A 0.000,B 0.000,C 90.000,E1 56.421} C_DIS
LIN {X -0.034,Y -540.930,Z 403.109,A 0.000,B 0.000,C 90.000,E1 55.548} C_DIS
LIN {X 0.028,Y -541.377,Z 403.104,A 0.000,B 0.000,C 90.000,E1 54.689} C_DIS
LIN {X 0.101,Y -541.469,Z 403.099,A 0.000,B 0.000,C 90.000,E1 53.829} C_DIS
LIN {X 0.152,Y -541.326,Z 403.096,A 0.000,B 0.000,C 90.000,E1 53.256} C_DIS
LIN {X -0.102,Y -540.921,Z 403.091,A 0.000,B 0.000,C 90.000,E1 52.431} C_DIS
LIN {X -0.106,Y -539.970,Z 403.085,A 0.000,B 0.000,C 90.000,E1 51.295} C_DIS
LIN {X -0.039,Y -538.773,Z 403.079,A 0.000,B 0.000,C 90.000,E1 50.150} C_DIS
LIN {X -0.065,Y -537.326,Z 403.072,A 0.000,B 0.000,C 90.000,E1 49.013} C_DIS
LIN {X 0.240,Y -535.238,Z 403.064,A 0.000,B 0.000,C 90.000,E1 47.553} C_DIS
LIN {X 0.016,Y -531.788,Z 403.052,A 0.000,B 0.000,C 90.000,E1 45.283} C_DIS
LIN {X 0.025,Y -528.305,Z 403.037,A 0.000,B 0.000,C 90.000,E1 42.690} C_DIS
LIN {X 0.040,Y -525.721,Z 403.026,A 0.000,B 0.000,C 90.000,E1 40.663} C_DIS
LIN {X 0.187,Y -523.973,Z 403.018,A 0.000,B 0.000,C 90.000,E1 39.197} C_DIS
LIN {X 0.308,Y -522.201,Z 403.010,A 0.000,B 0.000,C 90.000,E1 37.729} C_DIS
LIN {X 0.077,Y -520.340,Z 403.002,A 0.000,B 0.000,C 90.000,E1 36.297} C_DIS
LIN {X 0.173,Y -518.100,Z 402.992,A 0.000,B 0.000,C 90.000,E1 34.532} C_DIS
LIN {X -0.081,Y -515.739,Z 402.982,A 0.000,B 0.000,C 90.000,E1 32.801} C_DIS
LIN {X -0.148,Y -513.729,Z 402.974,A 0.000,B 0.000,C 90.000,E1 31.337} C_DIS
LIN {X -0.251,Y -511.033,Z 402.963,A 0.000,B 0.000,C 90.000,E1 29.283} C_DIS
LIN {X 0.102,Y -508.145,Z 402.949,A 0.000,B 0.000,C 90.000,E1 26.873} C_DIS
LIN {X -0.098,Y -505.480,Z 402.936,A 0.000,B 0.000,C 90.000,E1 24.515} C_DIS
LIN {X 0.139,Y -503.148,Z 402.923,A 0.000,B 0.000,C 90.000,E1 22.099} C_DIS
LIN {X 0.229,Y -501.439,Z 402.911,A 0.000,B 0.000,C 90.000,E1 19.993} C_DIS
LIN {X -0.218,Y -500.387,Z 402.903,A 0.000,B 0.000,C 90.000,E1 18.544} C_DIS
LIN {X -0.233,Y -499.022,Z 402.891,A 0.000,B 0.000,C 90.000,E1 16.441} C_DIS
LIN {X 0.004,Y -497.441,Z 402.876,A 0.000,B 0.000,C 90.000,E1 13.703} C_DIS
LIN {X 0.227,Y -496.329,Z 402.859,A 0.000,B 0.000,C 90.000,E1 10.658} C_DIS
LIN {X -0.243,Y -495.924,Z 402.844,A 0.000,B 0.000,C 90.000,E1 7.992} C_DIS
LIN {X -0.051,Y -496.405,Z 402.826,A 0.000,B 0.000,C 90.000,E1 4.645} C_DIS
LIN {X 0.109,Y -498.750,Z 402.802,A 0.000,B 0.000,C 90.000,E1 0.401} C_DIS
LIN {X 0.213,Y -501.830,Z 402.786,A 0.000,B 0.000,C 90.000,E1 357.364} C_DIS
LIN {X -0.251,Y -505.494,Z 402.771,A 0.000,B 0.000,C 90.000,E1 354.723} C_DIS
LIN {X -0.094,Y -510.845,Z 402.752,A 0.000,B 0.000,C 90.000,E1 351.432} C_DIS
LIN {X -0.005,Y -518.661,Z 402.731,A 0.000,B 0.000,C 90.000,E1 347.589} C_DIS
LIN {X -0.276,Y -525.117,Z 402.716,A 0.000,B 0.000,C 90.000,E1 344.991} C_DIS
LIN {X -0.250,Y -530.342,Z 402.705,A 0.000,B 0.000,C 90.000,E1 342.960} C_DIS
LIN {X -0.127,Y -534.968,Z 402.696,A 0.000,B 0.000,C 90.000,E1 341.221} C_DIS
LIN {X -0.022,Y -540.500,Z 402.685,A 0.000,B 0.000,C 90.000,E1 339.209} C_DIS
LIN {X -0.082,Y -546.208,Z 402.673,A 0.000,B 0.000,C 90.000,E1 337.230} C_DIS
LIN {X 0.219,Y -551.963,Z 402.663,A 0.000,B 0.000,C 90.000,E1 335.229} C_DIS
LIN {X -0.132,Y -557.065,Z 402.653,A 0.000,B 0.000,C 90.000,E1 333.589} C_DIS
LIN {X -0.274,Y -564.195,Z 402.641,A 0.000,B 0.000,C 90.000,E1 331.385} C_DIS
LIN {X 0.238,Y -570.476,Z 402.630,A 0.000,B 0.000,C 90.000,E1 329.410} C_DIS
LIN {X 0.090,Y -575.849,Z 402.621,A 0.000,B 0.000,C 90.000,E1 327.788} C_DIS
LIN {X 0.211,Y -580.293,Z 402.614,A 0.000,B 0.000,C 90.000,E1 326.421} C_DIS
LIN {X 0.144,Y -587.488,Z 402.602,A 0.000,B 0.000,C 90.000,E1 324.276} C_DIS
LIN {X -0.092,Y -590.147,Z 402.597,A 0.000,B 0.000,C 90.000,E1 323.497} C_DIS
LIN {X -0.090,Y -593.908,Z 402.591,A 0.000,B 0.000,C 90.000,E1 322.431} C_DIS
LIN {X 0.099,Y -600.444,Z 402.581,A 0.000,B 0.000,C 90.000,E1 320.561} C_DIS
LIN {X -0.234,Y -604.286,Z 402.575,A 0.000,B 0.000,C 90.000,E1 319.542} C_DIS
LIN {X -0.327,Y -608.979,Z 402.568,A 0.000,B 0.000,C 90.000,E1 318.243} C_DIS
LIN {X 0.076,Y -613.580,Z 402.561,A 0.000,B 0.000,C 90.000,E1 316.905} C_DIS
LIN {X -0.308,Y -618.124,Z 402.553,A 0.000,B 0.000,C 90.000,E1 315.648} C_DIS
LIN {X 0.272,Y -625.555,Z 402.542,A 0.000,B 0.000,C 90.000,E1 313.542} C_DIS
LIN {X 0.307,Y -632.000,Z 402.532,A 0.000,B 0.000,C 90.000,E1 311.757} C_DIS
LIN {X -0.200,Y -636.652,Z 402.525,A 0.000,B 0.000,C 90.000,E1 310.539} C_DIS
LIN {X -0.149,Y -641.072,Z 402.518,A 0.000,B 0.000,C 90.000,E1 309.277} C_DIS
LIN {X -0.024,Y -645.306,Z 402.511,A 0.000,B 0.000,C 90.000,E1 308.016} C_DIS
LIN {X -0.234,Y -649.329,Z 402.504,A 0.000,B 0.000,C 90.000,E1 306.790} C_DIS
LIN {X -0.316,Y -653.986,Z 402.496,A 0.000,B 0.000,C 90.000,E1 305.311} C_DIS
LIN {X 0.235,Y -658.369,Z 402.488,A 0.000,B 0.000,C 90.000,E1 303.785} C_DIS
LIN {X -0.042,Y -662.750,Z 402.480,A 0.000,B 0.000,C 90.000,E1 302.339} C_DIS
LIN {X 0.119,Y -667.708,Z 402.470,A 0.000,B 0.000,C 90.000,E1 300.620} C_DIS
LIN {X -0.085,Y -670.420,Z 402.465,A 0.000,B 0.000,C 90.000,E1 299.667} C_DIS
LIN {X -0.010,Y -672.864,Z 402.459,A 0.000,B 0.000,C 90.000,E1 298.693} C_DIS
LIN {X -0.078,Y -674.611,Z 402.455,A 0.000,B 0.000,C 90.000,E1 297.975} C_DIS
LIN {X 0.054,Y -676.689,Z 402.450,A 0.000,B 0.000,C 90.000,E1 297.001} C_DIS
LIN {X -0.312,Y -679.736,Z 402.442,A 0.000,B 0.000,C 90.000,E1 295.591} C_DIS
LIN {X 0.199,Y -681.456,Z 402.437,A 0.000,B 0.000,C 90.000,E1 294.591} C_DIS
LIN {X 0.115,Y -682.833,Z 402.431,A 0.000,B 0.000,C 90.000,E1 293.643} C_DIS
LIN {X -0.166,Y -683.535,Z 402.427,A 0.000,B 0.000,C 90.000,E1 292.950} C_DIS
LIN {X 0.187,Y -683.942,Z 402.423,A 0.000,B 0.000,C 90.000,E1 292.206} C_DIS
LIN {X -0.344,Y -684.170,Z 402.420,A 0.000,B 0.000,C 90.000,E1 291.535} C_DIS
LIN {X -0.027,Y -684.329,Z 402.414,A 0.000,B 0.000,C 90.000,E1 290.556} C_DIS
LIN {X 0.133,Y -684.246,Z 402.412,A 0.000,B 0.000,C 90.000,E1 290.066} C_DIS
LIN {X -0.235,Y -683.766,Z 402.405,A 0.000,B 0.000,C 90.000,E1 288.906} C_DIS
LIN {X 0.027,Y -682.899,Z 402.398,A 0.000,B 0.000,C 90.000,E1 287.692} C_DIS
LIN {X 0.097,Y -682.149,Z 402.393,A 0.000,B 0.000,C 90.000,E1 286.732} C_DIS
LIN {X -0.033,Y -681.277,Z 402.388,A 0.000,B 0.000,C 90.000,E1 285.788} C_DIS
LIN {X 0.083,Y -680.692,Z 402.385,A 0.000,B 0.000,C 90.000,E1 285.300} C_DIS
LIN {X -0.222,Y -678.041,Z 402.374,A 0.000,B 0.000,C 90.000,E1 283.411} C_DIS
LIN {X 0.020,Y -675.958,Z 402.366,A 0.000,B 0.000,C 90.000,E1 281.951} C_DIS
LIN {X -0.191,Y -674.628,Z 402.361,A 0.000,B 0.000,C 90.000,E1 281.007} C_DIS
LIN {X -0.204,Y -672.466,Z 402.352,A 0.000,B 0.000,C 90.000,E1 279.321} C_DIS
LIN {X 0.303,Y -670.543,Z 402.342,A 0.000,B 0.000,C 90.000,E1 277.587} C_DIS
LIN {X -0.068,Y -668.727,Z 402.332,A 0.000,B 0.000,C 90.000,E1 275.682} C_DIS
LIN {X 0.274,Y -667.382,Z 402.322,A 0.000,B 0.000,C 90.000,E1 273.955} C_DIS
LIN {X 0.192,Y -666.001,Z 402.310,A 0.000,B 0.000,C 90.000,E1 271.776} C_DIS
LIN {X 0.201,Y -665.511,Z 402.305,A 0.000,B 0.000,C 90.000,E1 270.802} C_DIS
LIN {X 0.207,Y -664.794,Z 402.299,A 0.000,B 0.000,C 90.000,E1 269.828} C_DIS
LIN {X 0.033,Y -663.578,Z 402.292,A 0.000,B 0.000,C 90.000,E1 268.625} C_DIS
LIN {X 0.030,Y -662.484,Z 402.287,A 0.000,B 0.000,C 90.000,E1 267.650} C_DIS
LIN {X 0.019,Y -661.219,Z 402.282,A 0.000,B 0.000,C 90.000,E1 266.674} C_DIS
LIN {X 0.315,Y -660.540,Z 402.279,A 0.000,B 0.000,C 90.000,E1 266.159} C_DIS
LIN {X 0.176,Y -660.301,Z 402.277,A 0.000,B 0.000,C 90.000,E1 265.927} C_DIS
LIN {X 0.270,Y -659.082,Z 402.273,A 0.000,B 0.000,C 90.000,E1 265.184} C_DIS
LIN {X 0.261,Y -657.139,Z 402.268,A 0.000,B 0.000,C 90.000,E1 264.204} C_DIS
LIN {X 0.233,Y -654.970,Z 402.263,A 0.000,B 0.000,C 90.000,E1 263.223} C_DIS
LIN {X -0.249,Y -653.237,Z 402.258,A 0.000,B 0.000,C 90.000,E1 262.527} C_DIS
LIN {X 0.181,Y -650.179,Z 402.252,A 0.000,B 0.000,C 90.000,E1 261.254} C_DIS
LIN {X -0.237,Y -646.013,Z 402.243,A 0.000,B 0.000,C 90.000,E1 259.803} C_DIS
LIN {X 0.165,Y -642.378,Z 402.236,A 0.000,B 0.000,C 90.000,E1 258.522} C_DIS
LIN {X 0.168,Y -639.412,Z 402.231,A 0.000,B 0.000,C 90.000,E1 257.521} C_DIS
LIN {X -0.205,Y -634.716,Z 402.222,A 0.000,B 0.000,C 90.000,E1 256.047} C_DIS
LIN {X -0.300,Y -631.402,Z 402.217,A 0.000,B 0.000,C 90.000,E1 255.046} C_DIS
LIN {X 0.325,Y -627.882,Z 402.211,A 0.000,B 0.000,C 90.000,E1 253.976} C_DIS
LIN {X 0.087,Y -623.277,Z 402.204,A 0.000,B 0.000,C 90.000,E1 252.725} C_DIS
LIN {X 0.183,Y -619.455,Z 402.198,A 0.000,B 0.000,C 90.000,E1 251.692} C_DIS
LIN {X -0.006,Y -614.593,Z 402.191,A 0.000,B 0.000,C 90.000,E1 250.423} C_DIS
LIN {X -0.022,Y -610.594,Z 402.186,A 0.000,B 0.000,C 90.000,E1 249.390} C_DIS
LIN {X 0.123,Y -606.416,Z 402.180,A 0.000,B 0.000,C 90.000,E1 248.337} C_DIS
LIN {X -0.086,Y -601.069,Z 402.173,A 0.000,B 0.000,C 90.000,E1 247.050} C_DIS
LIN {X 0.205,Y -593.319,Z 402.162,A 0.000,B 0.000,C 90.000,E1 245.177} C_DIS
LIN {X 0.126,Y -586.566,Z 402.153,A 0.000,B 0.000,C 90.000,E1 243.589} C_DIS
LIN {X 0.036,Y -578.758,Z 402.143,A 0.000,B 0.000,C 90.000,E1 241.719} C_DIS
LIN {X -0.144,Y -573.274,Z 402.135,A 0.000,B 0.000,C 90.000,E1 240.383} C_DIS
LIN {X -0.070,Y -563.792,Z 402.122,A 0.000,B 0.000,C 90.000,E1 237.916} C_DIS
LIN {X 0.291,Y -554.837,Z 402.108,A 0.000,B 0.000,C 90.000,E1 235.388} C_DIS
LIN {X -0.130,Y -550.067,Z 402.100,A 0.000,B 0.000,C 90.000,E1 234.036} C_DIS
LIN {X -0.149,Y -544.345,Z 402.091,A 0.000,B 0.000,C 90.000,E1 232.351} C_DIS
LIN {X -0.045,Y -537.651,Z 402.080,A 0.000,B 0.000,C 90.000,E1 230.356} C_DIS
LIN {X -0.301,Y -527.524,Z 402.062,A 0.000,B 0.000,C 90.000,E1 227.229} C_DIS
LIN {X -0.259,Y -522.250,Z 402.053,A 0.000,B 0.000,C 90.000,E1 225.486} C_DIS
LIN {X 0.025,Y -517.012,Z 402.043,A 0.000,B 0.000,C 90.000,E1 223.704} C_DIS
LIN {X -0.262,Y -511.038,Z 402.031,A 0.000,B 0.000,C 90.000,E1 221.676} C_DIS
LIN {X -0.042,Y -504.516,Z 402.018,A 0.000,B 0.000,C 90.000,E1 219.277} C_DIS
LIN {X 0.182,Y -499.051,Z 402.007,A 0.000,B 0.000,C 90.000,E1 217.156} C_DIS
LIN {X -0.337,Y -493.715,Z 401.995,A 0.000,B 0.000,C 90.000,E1 215.105} C_DIS
LIN {X -0.017,Y -489.367,Z 401.985,A 0.000,B 0.000,C 90.000,E1 213.245} C_DIS
LIN {X -0.243,Y -484.403,Z 401.973,A 0.000,B 0.000,C 90.000,E1 211.131} C_DIS
LIN {X -0.027,Y -479.423,Z 401.961,A 0.000,B 0.000,C 90.000,E1 208.949} C_DIS
LIN {X 0.089,Y -475.815,Z 401.952,A 0.000,B 0.000,C 90.000,E1 207.385} C_DIS
LIN {X -0.082,Y -472.146,Z 401.944,A 0.000,B 0.000,C 90.000,E1 205.848} C_DIS
LIN {X 0.097,Y -468.328,Z 401.935,A 0.000,B 0.000,C 90.000,E1 204.259} C_DIS
LIN {X -0.059,Y -463.724,Z 401.924,A 0.000,B 0.000,C 90.000,E1 202.386} C_DIS
LIN {X 0.015,Y -459.975,Z 401.916,A 0.000,B 0.000,C 90.000,E1 200.791} C_DIS
LIN {X 0.001,Y -454.295,Z 401.901,A 0.000,B 0.000,C 90.000,E1 198.236} C_DIS
LIN {X 0.093,Y -449.743,Z 401.889,A 0.000,B 0.000,C 90.000,E1 195.969} C_DIS
LIN {X -0.033,Y -444.414,Z 401.873,A 0.000,B 0.000,C 90.000,E1 193.063} C_DIS
LIN {X -0.135,Y -442.206,Z 401.865,A 0.000,B 0.000,C 90.000,E1 191.771} C_DIS
LIN {X 0.101,Y -438.533,Z 401.853,A 0.000,B 0.000,C 90.000,E1 189.443} C_DIS
LIN {X 0.172,Y -435.191,Z 401.840,A 0.000,B 0.000,C 90.000,E1 187.125} C_DIS
LIN {X -0.197,Y -431.502,Z 401.823,A 0.000,B 0.000,C 90.000,E1 184.188} C_DIS
LIN {X 0.101,Y -428.514,Z 401.806,A 0.000,B 0.000,C 90.000,E1 181.146} C_DIS
LIN {X 0.201,Y -425.561,Z 401.779,A 0.000,B 0.000,C 90.000,E1 176.102} C_DIS
LIN {X -0.054,Y -424.916,Z 401.762,A 0.000,B 0.000,C 90.000,E1 173.109} C_DIS
LIN {X -0.191,Y -426.188,Z 401.730,A 0.000,B 0.000,C 90.000,E1 167.409} C_DIS
LIN {X 0.153,Y -429.674,Z 401.704,A 0.000,B 0.000,C 90.000,E1 162.670} C_DIS
LIN {X -0.208,Y -434.222,Z 401.682,A 0.000,B 0.000,C 90.000,E1 158.720} C_DIS
LIN {X 0.072,Y -440.093,Z 401.660,A 0.000,B 0.000,C 90.000,E1 154.717} C_DIS
LIN {X 0.117,Y -446.106,Z 401.641,A 0.000,B 0.000,C 90.000,E1 151.435} C_DIS
LIN {X -0.130,Y -451.698,Z 401.627,A 0.000,B 0.000,C 90.000,E1 148.869} C_DIS
LIN {X -0.028,Y -459.742,Z 401.609,A 0.000,B 0.000,C 90.000,E1 145.642} C_DIS
LIN {X 0.213,Y -465.182,Z 401.599,A 0.000,B 0.000,C 90.000,E1 143.703} C_DIS
LIN {X -0.124,Y -471.948,Z 401.586,A 0.000,B 0.000,C 90.000,E1 141.537} C_DIS
LIN {X -0.154,Y -478.011,Z 401.576,A 0.000,B 0.000,C 90.000,E1 139.666} C_DIS
LIN {X 0.147,Y -483.077,Z 401.567,A 0.000,B 0.000,C 90.000,E1 138.081} C_DIS
LIN {X 0.034,Y -486.894,Z 401.560,A 0.000,B 0.000,C 90.000,E1 136.863} C_DIS
LIN {X 0.117,Y -491.409,Z 401.552,A 0.000,B 0.000,C 90.000,E1 135.324} C_DIS
LIN {X -0.068,Y -493.868,Z 401.547,A 0.000,B 0.000,C 90.000,E1 134.433} C_DIS
LIN {X -0.228,Y -496.174,Z 401.542,A 0.000,B 0.000,C 90.000,E1 133.542} C_DIS
LIN {X -0.005,Y -498.265,Z 401.537,A 0.000,B 0.000,C 90.000,E1 132.609} C_DIS
LIN {X 0.245,Y -500.090,Z 401.532,A 0.000,B 0.000,C 90.000,E1 131.676} C_DIS
LIN {X 0.185,Y -501.620,Z 401.527,A 0.000,B 0.000,C 90.000,E1 130.782} C_DIS
LIN {X 0.266,Y -502.501,Z 401.523,A 0.000,B 0.000,C 90.000,E1 130.172} C_DIS
LIN {X 0.122,Y -503.774,Z 401.517,A 0.000,B 0.000,C 90.000,E1 128.991} C_DIS
LIN {X 0.104,Y -504.232,Z 401.512,A 0.000,B 0.000,C 90.000,E1 128.096} C_DIS
LIN {X -0.222,Y -504.054,Z 401.507,A 0.000,B 0.000,C 90.000,E1 127.237} C_DIS
LIN {X 0.157,Y -503.281,Z 401.502,A 0.000,B 0.000,C 90.000,E1 126.297} C_DIS
LIN {X -0.181,Y -502.190,Z 401.497,A 0.000,B 0.000,C 90.000,E1 125.438} C_DIS
LIN {X -0.122,Y -500.710,Z 401.492,A 0.000,B 0.000,C 90.000,E1 124.532} C_DIS
LIN {X 0.046,Y -499.601,Z 401.488,A 0.000,B 0.000,C 90.000,E1 123.913} C_DIS
LIN {X 0.074,Y -497.333,Z 401.483,A 0.000,B 0.000,C 90.000,E1 123.007} C_DIS
LIN {X -0.194,Y -494.732,Z 401.478,A 0.000,B 0.000,C 90.000,E1 122.133} C_DIS
LIN {X 0.077,Y -493.830,Z 401.477,A 0.000,B 0.000,C 90.000,E1 121.799} C_DIS
LIN {X -0.227,Y -490.636,Z 401.472,A 0.000,B 0.000,C 90.000,E1 120.924} C_DIS
LIN {X 0.033,Y -488.367,Z 401.468,A 0.000,B 0.000,C 90.000,E1 120.285} C_DIS
LIN {X 0.096,Y -484.650,Z 401.463,A 0.000,B 0.000,C 90.000,E1 119.361} C_DIS
LIN {X 0.116,Y -480.088,Z 401.457,A 0.000,B 0.000,C 90.000,E1 118.281} C_DIS
LIN {X 0.029,Y -474.432,Z 401.450,A 0.000,B 0.000,C 90.000,E1 117.052} C_DIS
LIN {X -0.164,Y -467.721,Z 401.443,A 0.000,B 0.000,C 90.000,E1 115.668} C_DIS
LIN {X -0.094,Y -460.117,Z 401.434,A 0.000,B 0.000,C 90.000,E1 114.079} C_DIS
LIN {X 0.056,Y -452.404,Z 401.425,A 0.000,B 0.000,C 90.000,E1 112.461} C_DIS
LIN {X 0.188,Y -450.983,Z 401.423,A 0.000,B 0.000,C 90.000,E1 112.153} C_DIS
LIN {X 0.148,Y -450.977,Z 401.423,A 0.000,B 0.000,C 90.000,E1 112.153} C_DIS
LIN {X 0.045,Y -457.034,Z 401.411,A 0.000,B 0.000,C 90.000,E1 109.885} C_DIS
LIN {X 0.193,Y -458.871,Z 401.405,A 0.000,B 0.000,C 90.000,E1 108.906} C_DIS
LIN {X -0.150,Y -467.231,Z 401.384,A 0.000,B 0.000,C 90.000,E1 105.134} C_DIS
LIN {X 0.226,Y -467.942,Z 401.382,A 0.000,B 0.000,C 90.000,E1 104.773} C_DIS
LIN {X 0.191,Y -476.159,Z 401.356,A 0.000,B 0.000,C 90.000,E1 100.074} C_DIS
LIN {X -0.079,Y -482.069,Z 401.330,A 0.000,B 0.000,C 90.000,E1 95.454} C_DIS
LIN {X 0.197,Y -485.493,Z 401.305,A 0.000,B 0.000,C 90.000,E1 90.802} C_DIS
LIN {X 0.229,Y -486.385,Z 401.281,A 0.000,B 0.000,C 90.000,E1 86.502} C_DIS
LIN {X 0.054,Y -486.362,Z 401.279,A 0.000,B 0.000,C 90.000,E1 86.216} C_DIS
LIN {X 0.137,Y -484.688,Z 401.253,A 0.000,B 0.000,C 90.000,E1 81.602} C_DIS
LIN {X 0.037,Y -480.615,Z 401.228,A 0.000,B 0.000,C 90.000,E1 76.992} C_DIS
LIN {X -0.106,Y -480.269,Z 401.226,A 0.000,B 0.000,C 90.000,E1 76.700} C_DIS
LIN {X 0.250,Y -474.096,Z 401.200,A 0.000,B 0.000,C 90.000,E1 72.000} C_DIS
LIN {X -0.033,Y -470.389,Z 401.190,A 0.000,B 0.000,C 90.000,E1 70.115} C_DIS
LIN {X -0.073,Y -470.421,Z 401.190,A 0.000,B 0.000,C 90.000,E1 70.115} C_DIS
LIN {X 0.031,Y -479.499,Z 401.183,A 0.000,B 0.000,C 90.000,E1 68.901} C_DIS
LIN {X -0.201,Y -487.503,Z 401.177,A 0.000,B 0.000,C 90.000,E1 67.847} C_DIS
LIN {X -0.220,Y -493.087,Z 401.173,A 0.000,B 0.000,C 90.000,E1 67.102} C_DIS
LIN {X 0.069,Y -496.520,Z 401.170,A 0.000,B 0.000,C 90.000,E1 66.613} C_DIS
LIN {X -0.214,Y -502.935,Z 401.165,A 0.000,B 0.000,C 90.000,E1 65.741} C_DIS
LIN {X 0.150,Y -507.112,Z 401.162,A 0.000,B 0.000,C 90.000,E1 65.101} C_DIS
LIN {X -0.024,Y -512.702,Z 401.157,A 0.000,B 0.000,C 90.000,E1 64.229} C_DIS
LIN {X 0.082,Y -517.985,Z 401.152,A 0.000,B 0.000,C 90.000,E1 63.332} C_DIS
LIN {X -0.054,Y -521.935,Z 401.148,A 0.000,B 0.000,C 90.000,E1 62.615} C_DIS
LIN {X -0.150,Y -525.394,Z 401.144,A 0.000,B 0.000,C 90.000,E1 61.897} C_DIS
LIN {X 0.093,Y -527.357,Z 401.141,A 0.000,B 0.000,C 90.000,E1 61.435} C_DIS
LIN {X -0.108,Y -530.691,Z 401.137,A 0.000,B 0.000,C 90.000,E1 60.589} C_DIS
LIN {X 0.017,Y -532.720,Z 401.133,A 0.000,B 0.000,C 90.000,E1 59.999} C_DIS
LIN {X 0.156,Y -534.577,Z 401.130,A 0.000,B 0.000,C 90.000,E1 59.410} C_DIS
LIN {X 0.296,Y -536.865,Z 401.125,A 0.000,B 0.000,C 90.000,E1 58.535} C_DIS
LIN {X 0.006,Y -538.238,Z 401.122,A 0.000,B 0.000,C 90.000,E1 57.995} C_DIS
LIN {X -0.277,Y -539.415,Z 401.119,A 0.000,B 0.000,C 90.000,E1 57.454} C_DIS
LIN {X -0.086,Y -540.728,Z 401.114,A 0.000,B 0.000,C 90.000,E1 56.580} C_DIS
LIN {X -0.031,Y -541.657,Z 401.110,A 0.000,B 0.000,C 90.000,E1 55.722} C_DIS
LIN {X -0.292,Y -542.117,Z 401.106,A 0.000,B 0.000,C 90.000,E1 55.182} C_DIS
LIN {X 0.228,Y -542.453,Z 401.102,A 0.000,B 0.000,C 90.000,E1 54.276} C_DIS
LIN {X 0.311,Y -542.385,Z 401.097,A 0.000,B 0.000,C 90.000,E1 53.417} C_DIS
LIN {X -0.035,Y -542.107,Z 401.092,A 0.000,B 0.000,C 90.000,E1 52.603} C_DIS
LIN {X 0.073,Y -541.202,Z 401.086,A 0.000,B 0.000,C 90.000,E1 51.457} C_DIS
LIN {X -0.259,Y -540.092,Z 401.080,A 0.000,B 0.000,C 90.000,E1 50.356} C_DIS
LIN {X 0.145,Y -538.664,Z 401.073,A 0.000,B 0.000,C 90.000,E1 49.175} C_DIS
LIN {X -0.286,Y -537.005,Z 401.067,A 0.000,B 0.000,C 90.000,E1 48.081} C_DIS
LIN {X -0.021,Y -534.376,Z 401.057,A 0.000,B 0.000,C 90.000,E1 46.338} C_DIS
LIN {X -0.226,Y -531.468,Z 401.046,A 0.000,B 0.000,C 90.000,E1 44.352} C_DIS
LIN {X -0.087,Y -529.196,Z 401.037,A 0.000,B 0.000,C 90.000,E1 42.609} C_DIS
LIN {X 0.351,Y -526.613,Z 401.025,A 0.000,B 0.000,C 90.000,E1 40.539} C_DIS
LIN {X 0.150,Y -525.232,Z 401.019,A 0.000,B 0.000,C 90.000,E1 39.402} C_DIS
LIN {X -0.032,Y -523.445,Z 401.011,A 0.000,B 0.000,C 90.000,E1 37.971} C_DIS
LIN {X 0.077,Y -521.599,Z 401.003,A 0.000,B 0.000,C 90.000,E1 36.503} C_DIS
LIN {X 0.200,Y -519.334,Z 400.993,A 0.000,B 0.000,C 90.000,E1 34.739} C_DIS
LIN {X -0.028,Y -517.005,Z 400.983,A 0.000,B 0.000,C 90.000,E1 33.007} C_DIS
LIN {X 0.277,Y -515.401,Z 400.977,A 0.000,B 0.000,C 90.000,E1 31.799} C_DIS
LIN {X 0.112,Y -512.295,Z 400.964,A 0.000,B 0.000,C 90.000,E1 29.461} C_DIS
LIN {X -0.196,Y -509.411,Z 400.951,A 0.000,B 0.000,C 90.000,E1 27.129} C_DIS
LIN {X 0.104,Y -506.732,Z 400.937,A 0.000,B 0.000,C 90.000,E1 24.719} C_DIS
LIN {X 0.201,Y -504.083,Z 400.923,A 0.000,B 0.000,C 90.000,E1 22.025} C_DIS
LIN {X 0.212,Y -502.189,Z 400.909,A 0.000,B 0.000,C 90.000,E1 19.631} C_DIS
LIN {X -0.237,Y -500.721,Z 400.898,A 0.000,B 0.000,C 90.000,E1 17.583} C_DIS
LIN {X -0.218,Y -499.771,Z 400.889,A 0.000,B 0.000,C 90.000,E1 16.079} C_DIS
LIN {X 0.000,Y -498.430,Z 400.876,A 0.000,B 0.000,C 90.000,E1 13.647} C_DIS
LIN {X -0.139,Y -497.467,Z 400.861,A 0.000,B 0.000,C 90.000,E1 10.950} C_DIS
LIN {X 0.169,Y -497.088,Z 400.849,A 0.000,B 0.000,C 90.000,E1 8.803} C_DIS
LIN {X -0.175,Y -497.379,Z 400.829,A 0.000,B 0.000,C 90.000,E1 5.220} C_DIS
LIN {X -0.187,Y -499.094,Z 400.809,A 0.000,B 0.000,C 90.000,E1 1.604} C_DIS
LIN {X -0.251,Y -503.113,Z 400.786,A 0.000,B 0.000,C 90.000,E1 357.421} C_DIS
LIN {X -0.171,Y -506.784,Z 400.771,A 0.000,B 0.000,C 90.000,E1 354.723} C_DIS
LIN {X 0.040,Y -512.190,Z 400.752,A 0.000,B 0.000,C 90.000,E1 351.432} C_DIS
LIN {X 0.192,Y -520.710,Z 400.730,A 0.000,B 0.000,C 90.000,E1 347.297} C_DIS
LIN {X -0.026,Y -526.536,Z 400.717,A 0.000,B 0.000,C 90.000,E1 344.991} C_DIS
LIN {X 0.040,Y -531.800,Z 400.705,A 0.000,B 0.000,C 90.000,E1 342.960} C_DIS
LIN {X 0.197,Y -536.448,Z 400.696,A 0.000,B 0.000,C 90.000,E1 341.221} C_DIS
LIN {X -0.162,Y -542.015,Z 400.685,A 0.000,B 0.000,C 90.000,E1 339.263} C_DIS
LIN {X -0.179,Y -547.704,Z 400.674,A 0.000,B 0.000,C 90.000,E1 337.283} C_DIS
LIN {X 0.168,Y -553.462,Z 400.663,A 0.000,B 0.000,C 90.000,E1 335.281} C_DIS
LIN {X 0.144,Y -559.449,Z 400.652,A 0.000,B 0.000,C 90.000,E1 333.332} C_DIS
LIN {X 0.262,Y -565.676,Z 400.641,A 0.000,B 0.000,C 90.000,E1 331.385} C_DIS
LIN {X 0.035,Y -571.955,Z 400.631,A 0.000,B 0.000,C 90.000,E1 329.488} C_DIS
LIN {X -0.089,Y -577.344,Z 400.621,A 0.000,B 0.000,C 90.000,E1 327.867} C_DIS
LIN {X 0.052,Y -581.785,Z 400.614,A 0.000,B 0.000,C 90.000,E1 326.501} C_DIS
LIN {X 0.167,Y -588.092,Z 400.604,A 0.000,B 0.000,C 90.000,E1 324.609} C_DIS
LIN {X -0.040,Y -594.514,Z 400.593,A 0.000,B 0.000,C 90.000,E1 322.763} C_DIS
LIN {X 0.023,Y -600.111,Z 400.584,A 0.000,B 0.000,C 90.000,E1 321.170} C_DIS
LIN {X 0.325,Y -604.895,Z 400.577,A 0.000,B 0.000,C 90.000,E1 319.828} C_DIS
LIN {X -0.341,Y -610.537,Z 400.568,A 0.000,B 0.000,C 90.000,E1 318.324} C_DIS
LIN {X 0.088,Y -615.162,Z 400.561,A 0.000,B 0.000,C 90.000,E1 316.986} C_DIS
LIN {X -0.115,Y -618.832,Z 400.555,A 0.000,B 0.000,C 90.000,E1 315.972} C_DIS
LIN {X -0.122,Y -624.268,Z 400.547,A 0.000,B 0.000,C 90.000,E1 314.433} C_DIS
LIN {X 0.227,Y -628.044,Z 400.541,A 0.000,B 0.000,C 90.000,E1 313.380} C_DIS
LIN {X 0.319,Y -634.528,Z 400.531,A 0.000,B 0.000,C 90.000,E1 311.595} C_DIS
LIN {X -0.049,Y -638.258,Z 400.526,A 0.000,B 0.000,C 90.000,E1 310.620} C_DIS
LIN {X 0.034,Y -642.715,Z 400.519,A 0.000,B 0.000,C 90.000,E1 309.358} C_DIS
LIN {X 0.188,Y -646.928,Z 400.512,A 0.000,B 0.000,C 90.000,E1 308.096} C_DIS
LIN {X 0.091,Y -650.171,Z 400.506,A 0.000,B 0.000,C 90.000,E1 307.111} C_DIS
LIN {X -0.109,Y -654.874,Z 400.498,A 0.000,B 0.000,C 90.000,E1 305.644} C_DIS
LIN {X 0.084,Y -659.301,Z 400.490,A 0.000,B 0.000,C 90.000,E1 304.151} C_DIS
LIN {X 0.193,Y -663.671,Z 400.482,A 0.000,B 0.000,C 90.000,E1 302.673} C_DIS
LIN {X 0.080,Y -667.264,Z 400.475,A 0.000,B 0.000,C 90.000,E1 301.465} C_DIS
LIN {X -0.130,Y -670.074,Z 400.470,A 0.000,B 0.000,C 90.000,E1 300.512} C_DIS
LIN {X 0.186,Y -671.476,Z 400.467,A 0.000,B 0.000,C 90.000,E1 300.001} C_DIS
LIN {X 0.103,Y -673.378,Z 400.463,A 0.000,B 0.000,C 90.000,E1 299.283} C_DIS
LIN {X -0.373,Y -675.685,Z 400.457,A 0.000,B 0.000,C 90.000,E1 298.359} C_DIS
LIN {X -0.229,Y -677.857,Z 400.452,A 0.000,B 0.000,C 90.000,E1 297.385} C_DIS
LIN {X 0.351,Y -679.311,Z 400.448,A 0.000,B 0.000,C 90.000,E1 296.616} C_DIS
LIN {X 0.240,Y -681.199,Z 400.443,A 0.000,B 0.000,C 90.000,E1 295.668} C_DIS
LIN {X 0.157,Y -682.786,Z 400.437,A 0.000,B 0.000,C 90.000,E1 294.719} C_DIS
LIN {X 0.092,Y -684.091,Z 400.432,A 0.000,B 0.000,C 90.000,E1 293.770} C_DIS
LIN {X -0.177,Y -684.787,Z 400.428,A 0.000,B 0.000,C 90.000,E1 293.078} C_DIS
LIN {X 0.190,Y -685.194,Z 400.424,A 0.000,B 0.000,C 90.000,E1 292.333} C_DIS
LIN {X -0.077,Y -685.356,Z 400.420,A 0.000,B 0.000,C 90.000,E1 291.642} C_DIS
LIN {X 0.247,Y -685.377,Z 400.415,A 0.000,B 0.000,C 90.000,E1 290.663} C_DIS
LIN {X -0.269,Y -685.000,Z 400.411,A 0.000,B 0.000,C 90.000,E1 289.993} C_DIS
LIN {X -0.176,Y -684.431,Z 400.406,A 0.000,B 0.000,C 90.000,E1 289.033} C_DIS
LIN {X -0.049,Y -683.785,Z 400.402,A 0.000,B 0.000,C 90.000,E1 288.308} C_DIS
LIN {X 0.071,Y -682.991,Z 400.398,A 0.000,B 0.000,C 90.000,E1 287.583} C_DIS
LIN {X 0.040,Y -682.663,Z 400.396,A 0.000,B 0.000,C 90.000,E1 287.347} C_DIS
LIN {X 0.179,Y -682.305,Z 400.394,A 0.000,B 0.000,C 90.000,E1 286.858} C_DIS
LIN {X 0.241,Y -681.282,Z 400.388,A 0.000,B 0.000,C 90.000,E1 285.898} C_DIS
LIN {X 0.174,Y -680.729,Z 400.386,A 0.000,B 0.000,C 90.000,E1 285.426} C_DIS
LIN {X -0.121,Y -678.031,Z 400.375,A 0.000,B 0.000,C 90.000,E1 283.536} C_DIS
LIN {X 0.319,Y -676.261,Z 400.369,A 0.000,B 0.000,C 90.000,E1 282.299} C_DIS
LIN {X -0.076,Y -674.489,Z 400.362,A 0.000,B 0.000,C 90.000,E1 281.130} C_DIS
LIN {X 0.266,Y -671.383,Z 400.348,A 0.000,B 0.000,C 90.000,E1 278.690} C_DIS
LIN {X 0.236,Y -668.573,Z 400.334,A 0.000,B 0.000,C 90.000,E1 276.030} C_DIS
LIN {X -0.244,Y -667.154,Z 400.323,A 0.000,B 0.000,C 90.000,E1 274.131} C_DIS
LIN {X -0.310,Y -665.878,Z 400.311,A 0.000,B 0.000,C 90.000,E1 271.949} C_DIS
LIN {X 0.219,Y -665.235,Z 400.304,A 0.000,B 0.000,C 90.000,E1 270.688} C_DIS
LIN {X 0.222,Y -664.478,Z 400.299,A 0.000,B 0.000,C 90.000,E1 269.714} C_DIS
LIN {X 0.214,Y -663.595,Z 400.293,A 0.000,B 0.000,C 90.000,E1 268.740} C_DIS
LIN {X 0.210,Y -662.709,Z 400.288,A 0.000,B 0.000,C 90.000,E1 267.764} C_DIS
LIN {X 0.183,Y -660.687,Z 400.277,A 0.000,B 0.000,C 90.000,E1 265.812} C_DIS
LIN {X 0.335,Y -659.615,Z 400.273,A 0.000,B 0.000,C 90.000,E1 265.065} C_DIS
LIN {X -0.182,Y -658.297,Z 400.269,A 0.000,B 0.000,C 90.000,E1 264.375} C_DIS
LIN {X 0.254,Y -655.729,Z 400.262,A 0.000,B 0.000,C 90.000,E1 263.109} C_DIS
LIN {X 0.204,Y -653.467,Z 400.256,A 0.000,B 0.000,C 90.000,E1 262.129} C_DIS
LIN {X 0.217,Y -651.074,Z 400.251,A 0.000,B 0.000,C 90.000,E1 261.141} C_DIS
LIN {X -0.048,Y -647.682,Z 400.244,A 0.000,B 0.000,C 90.000,E1 259.926} C_DIS
LIN {X -0.258,Y -644.139,Z 400.237,A 0.000,B 0.000,C 90.000,E1 258.701} C_DIS
LIN {X 0.234,Y -640.471,Z 400.230,A 0.000,B 0.000,C 90.000,E1 257.409} C_DIS
LIN {X -0.125,Y -635.809,Z 400.222,A 0.000,B 0.000,C 90.000,E1 255.936} C_DIS
LIN {X -0.213,Y -632.516,Z 400.216,A 0.000,B 0.000,C 90.000,E1 254.936} C_DIS
LIN {X -0.182,Y -629.009,Z 400.211,A 0.000,B 0.000,C 90.000,E1 253.921} C_DIS
LIN {X -0.217,Y -624.426,Z 400.204,A 0.000,B 0.000,C 90.000,E1 252.653} C_DIS
LIN {X 0.072,Y -619.621,Z 400.196,A 0.000,B 0.000,C 90.000,E1 251.348} C_DIS
LIN {X 0.081,Y -614.738,Z 400.189,A 0.000,B 0.000,C 90.000,E1 250.061} C_DIS
LIN {X 0.062,Y -610.686,Z 400.184,A 0.000,B 0.000,C 90.000,E1 249.028} C_DIS
LIN {X 0.151,Y -605.403,Z 400.176,A 0.000,B 0.000,C 90.000,E1 247.720} C_DIS
LIN {X 0.227,Y -601.046,Z 400.171,A 0.000,B 0.000,C 90.000,E1 246.666} C_DIS
LIN {X 0.068,Y -594.406,Z 400.162,A 0.000,B 0.000,C 90.000,E1 245.101} C_DIS
LIN {X 0.021,Y -587.674,Z 400.153,A 0.000,B 0.000,C 90.000,E1 243.512} C_DIS
LIN {X -0.033,Y -579.857,Z 400.142,A 0.000,B 0.000,C 90.000,E1 241.641} C_DIS
LIN {X 0.026,Y -574.376,Z 400.135,A 0.000,B 0.000,C 90.000,E1 240.284} C_DIS
LIN {X -0.070,Y -564.924,Z 400.121,A 0.000,B 0.000,C 90.000,E1 237.837} C_DIS
LIN {X 0.019,Y -556.020,Z 400.108,A 0.000,B 0.000,C 90.000,E1 235.341} C_DIS
LIN {X -0.322,Y -550.324,Z 400.098,A 0.000,B 0.000,C 90.000,E1 233.703} C_DIS
LIN {X -0.011,Y -544.638,Z 400.089,A 0.000,B 0.000,C 90.000,E1 231.984} C_DIS
LIN {X 0.084,Y -538.877,Z 400.079,A 0.000,B 0.000,C 90.000,E1 230.275} C_DIS
LIN {X 0.294,Y -529.635,Z 400.064,A 0.000,B 0.000,C 90.000,E1 227.391} C_DIS
LIN {X 0.007,Y -524.364,Z 400.054,A 0.000,B 0.000,C 90.000,E1 225.688} C_DIS
LIN {X -0.034,Y -519.097,Z 400.044,A 0.000,B 0.000,C 90.000,E1 223.947} C_DIS
LIN {X -0.007,Y -512.251,Z 400.031,A 0.000,B 0.000,C 90.000,E1 221.595} C_DIS
LIN {X 0.244,Y -505.709,Z 400.018,A 0.000,B 0.000,C 90.000,E1 219.197} C_DIS
LIN {X -0.209,Y -500.239,Z 400.006,A 0.000,B 0.000,C 90.000,E1 217.156} C_DIS
LIN {X -0.005,Y -494.914,Z 399.995,A 0.000,B 0.000,C 90.000,E1 215.025} C_DIS
LIN {X -0.075,Y -490.529,Z 399.985,A 0.000,B 0.000,C 90.000,E1 213.214} C_DIS
LIN {X 0.130,Y -485.569,Z 399.973,A 0.000,B 0.000,C 90.000,E1 211.052} C_DIS
LIN {X 0.156,Y -481.330,Z 399.962,A 0.000,B 0.000,C 90.000,E1 209.205} C_DIS
LIN {X -0.144,Y -477.006,Z 399.952,A 0.000,B 0.000,C 90.000,E1 207.385} C_DIS
LIN {X 0.166,Y -474.098,Z 399.945,A 0.000,B 0.000,C 90.000,E1 206.104} C_DIS
LIN {X -0.044,Y -470.286,Z 399.936,A 0.000,B 0.000,C 90.000,E1 204.567} C_DIS
LIN {X -0.157,Y -465.723,Z 399.926,A 0.000,B 0.000,C 90.000,E1 202.695} C_DIS
LIN {X -0.117,Y -461.186,Z 399.915,A 0.000,B 0.000,C 90.000,E1 200.791} C_DIS
LIN {X -0.093,Y -455.497,Z 399.901,A 0.000,B 0.000,C 90.000,E1 198.236} C_DIS
LIN {X -0.092,Y -450.265,Z 399.887,A 0.000,B 0.000,C 90.000,E1 195.662} C_DIS
LIN {X -0.052,Y -445.552,Z 399.873,A 0.000,B 0.000,C 90.000,E1 193.063} C_DIS
LIN {X -0.137,Y -443.323,Z 399.865,A 0.000,B 0.000,C 90.000,E1 191.771} C_DIS
LIN {X -0.185,Y -440.648,Z 399.856,A 0.000,B 0.000,C 90.000,E1 190.141} C_DIS
LIN {X 0.003,Y -438.630,Z 399.849,A 0.000,B 0.000,C 90.000,E1 188.803} C_DIS
LIN {X -0.202,Y -436.235,Z 399.840,A 0.000,B 0.000,C 90.000,E1 187.182} C_DIS
LIN {X -0.102,Y -432.527,Z 399.823,A 0.000,B 0.000,C 90.000,E1 184.188} C_DIS
LIN {X -0.198,Y -429.500,Z 399.807,A 0.000,B 0.000,C 90.000,E1 181.203} C_DIS
LIN {X -0.038,Y -426.507,Z 399.779,A 0.000,B 0.000,C 90.000,E1 176.159} C_DIS
LIN {X 0.165,Y -425.862,Z 399.762,A 0.000,B 0.000,C 90.000,E1 173.109} C_DIS
LIN {X 0.090,Y -427.091,Z 399.730,A 0.000,B 0.000,C 90.000,E1 167.409} C_DIS
LIN {X 0.097,Y -431.209,Z 399.700,A 0.000,B 0.000,C 90.000,E1 162.054} C_DIS
LIN {X -0.005,Y -435.534,Z 399.680,A 0.000,B 0.000,C 90.000,E1 158.411} C_DIS
LIN {X -0.059,Y -441.529,Z 399.658,A 0.000,B 0.000,C 90.000,E1 154.460} C_DIS
LIN {X 0.040,Y -447.654,Z 399.640,A 0.000,B 0.000,C 90.000,E1 151.179} C_DIS
LIN {X -0.020,Y -452.607,Z 399.627,A 0.000,B 0.000,C 90.000,E1 148.918} C_DIS
LIN {X -0.007,Y -461.567,Z 399.608,A 0.000,B 0.000,C 90.000,E1 145.388} C_DIS
LIN {X -0.108,Y -467.077,Z 399.597,A 0.000,B 0.000,C 90.000,E1 143.497} C_DIS
LIN {X -0.108,Y -473.968,Z 399.585,A 0.000,B 0.000,C 90.000,E1 141.295} C_DIS
LIN {X -0.191,Y -479.066,Z 399.576,A 0.000,B 0.000,C 90.000,E1 139.747} C_DIS
LIN {X 0.130,Y -484.158,Z 399.568,A 0.000,B 0.000,C 90.000,E1 138.162} C_DIS
LIN {X 0.218,Y -487.086,Z 399.563,A 0.000,B 0.000,C 90.000,E1 137.229} C_DIS
LIN {X -0.195,Y -490.751,Z 399.556,A 0.000,B 0.000,C 90.000,E1 136.053} C_DIS
LIN {X -0.040,Y -493.412,Z 399.551,A 0.000,B 0.000,C 90.000,E1 135.121} C_DIS
LIN {X 0.331,Y -496.570,Z 399.544,A 0.000,B 0.000,C 90.000,E1 133.866} C_DIS
LIN {X -0.142,Y -498.779,Z 399.539,A 0.000,B 0.000,C 90.000,E1 133.014} C_DIS
LIN {X 0.117,Y -500.736,Z 399.534,A 0.000,B 0.000,C 90.000,E1 132.081} C_DIS
LIN {X -0.312,Y -502.377,Z 399.529,A 0.000,B 0.000,C 90.000,E1 131.229} C_DIS
LIN {X -0.136,Y -504.198,Z 399.522,A 0.000,B 0.000,C 90.000,E1 130.011} C_DIS
LIN {X -0.151,Y -505.174,Z 399.517,A 0.000,B 0.000,C 90.000,E1 129.116} C_DIS
LIN {X 0.240,Y -505.688,Z 399.512,A 0.000,B 0.000,C 90.000,E1 128.177} C_DIS
LIN {X 0.137,Y -505.747,Z 399.511,A 0.000,B 0.000,C 90.000,E1 127.890} C_DIS
LIN {X 0.133,Y -505.437,Z 399.506,A 0.000,B 0.000,C 90.000,E1 126.996} C_DIS
LIN {X 0.226,Y -504.623,Z 399.501,A 0.000,B 0.000,C 90.000,E1 126.091} C_DIS
LIN {X 0.012,Y -503.903,Z 399.497,A 0.000,B 0.000,C 90.000,E1 125.518} C_DIS
LIN {X 0.091,Y -502.490,Z 399.492,A 0.000,B 0.000,C 90.000,E1 124.612} C_DIS
LIN {X -0.142,Y -501.409,Z 399.489,A 0.000,B 0.000,C 90.000,E1 124.040} C_DIS
LIN {X 0.031,Y -500.048,Z 399.486,A 0.000,B 0.000,C 90.000,E1 123.420} C_DIS
LIN {X -0.077,Y -498.506,Z 399.482,A 0.000,B 0.000,C 90.000,E1 122.832} C_DIS
LIN {X 0.213,Y -494.896,Z 399.476,A 0.000,B 0.000,C 90.000,E1 121.592} C_DIS
LIN {X -0.081,Y -491.673,Z 399.471,A 0.000,B 0.000,C 90.000,E1 120.718} C_DIS
LIN {X 0.013,Y -488.183,Z 399.466,A 0.000,B 0.000,C 90.000,E1 119.795} C_DIS
LIN {X 0.065,Y -484.368,Z 399.460,A 0.000,B 0.000,C 90.000,E1 118.871} C_DIS
LIN {X -0.161,Y -480.349,Z 399.455,A 0.000,B 0.000,C 90.000,E1 117.975} C_DIS
LIN {X -0.009,Y -475.344,Z 399.449,A 0.000,B 0.000,C 90.000,E1 116.873} C_DIS
LIN {X 0.256,Y -469.385,Z 399.442,A 0.000,B 0.000,C 90.000,E1 115.591} C_DIS
LIN {X 0.157,Y -461.723,Z 399.434,A 0.000,B 0.000,C 90.000,E1 114.027} C_DIS
LIN {X 0.014,Y -455.516,Z 399.427,A 0.000,B 0.000,C 90.000,E1 112.770} C_DIS
LIN {X -0.012,Y -451.542,Z 399.422,A 0.000,B 0.000,C 90.000,E1 111.950} C_DIS
LIN {X -0.052,Y -451.542,Z 399.422,A 0.000,B 0.000,C 90.000,E1 111.950} C_DIS
LIN {X -0.239,Y -456.621,Z 399.411,A 0.000,B 0.000,C 90.000,E1 110.066} C_DIS
LIN {X 0.094,Y -457.441,Z 399.410,A 0.000,B 0.000,C 90.000,E1 109.704} C_DIS
LIN {X -0.254,Y -466.096,Z 399.387,A 0.000,B 0.000,C 90.000,E1 105.607} C_DIS
LIN {X -0.081,Y -467.667,Z 399.383,A 0.000,B 0.000,C 90.000,E1 104.954} C_DIS
LIN {X -0.093,Y -473.979,Z 399.362,A 0.000,B 0.000,C 90.000,E1 101.186} C_DIS
LIN {X -0.124,Y -475.882,Z 399.357,A 0.000,B 0.000,C 90.000,E1 100.254} C_DIS
LIN {X 0.183,Y -476.341,Z 399.355,A 0.000,B 0.000,C 90.000,E1 99.905} C_DIS
LIN {X 0.141,Y -481.850,Z 399.331,A 0.000,B 0.000,C 90.000,E1 95.568} C_DIS
LIN {X -0.013,Y -482.187,Z 399.329,A 0.000,B 0.000,C 90.000,E1 95.277} C_DIS
LIN {X -0.078,Y -485.348,Z 399.305,A 0.000,B 0.000,C 90.000,E1 90.974} C_DIS
LIN {X 0.231,Y -485.533,Z 399.304,A 0.000,B 0.000,C 90.000,E1 90.630} C_DIS
LIN {X -0.047,Y -486.338,Z 399.282,A 0.000,B 0.000,C 90.000,E1 86.674} C_DIS
LIN {X 0.088,Y -486.278,Z 399.278,A 0.000,B 0.000,C 90.000,E1 86.045} C_DIS
LIN {X -0.192,Y -484.694,Z 399.254,A 0.000,B 0.000,C 90.000,E1 81.781} C_DIS
LIN {X 0.156,Y -484.554,Z 399.253,A 0.000,B 0.000,C 90.000,E1 81.432} C_DIS
LIN {X 0.025,Y -480.493,Z 399.227,A 0.000,B 0.000,C 90.000,E1 76.825} C_DIS
LIN {X -0.078,Y -474.247,Z 399.201,A 0.000,B 0.000,C 90.000,E1 72.181} C_DIS
LIN {X -0.110,Y -473.768,Z 399.199,A 0.000,B 0.000,C 90.000,E1 71.873} C_DIS
LIN {X 0.011,Y -470.760,Z 399.191,A 0.000,B 0.000,C 90.000,E1 70.315} C_DIS
LIN {X -0.029,Y -470.779,Z 399.191,A 0.000,B 0.000,C 90.000,E1 70.315} C_DIS
LIN {X 0.163,Y -480.268,Z 399.184,A 0.000,B 0.000,C 90.000,E1 69.028} C_DIS
LIN {X 0.175,Y -489.385,Z 399.177,A 0.000,B 0.000,C 90.000,E1 67.794} C_DIS
LIN {X -0.182,Y -496.221,Z 399.172,A 0.000,B 0.000,C 90.000,E1 66.922} C_DIS
LIN {X -0.012,Y -502.622,Z 399.167,A 0.000,B 0.000,C 90.000,E1 65.997} C_DIS
LIN {X 0.164,Y -507.763,Z 399.163,A 0.000,B 0.000,C 90.000,E1 65.229} C_DIS
LIN {X -0.287,Y -512.416,Z 399.158,A 0.000,B 0.000,C 90.000,E1 64.537} C_DIS
LIN {X 0.158,Y -515.917,Z 399.155,A 0.000,B 0.000,C 90.000,E1 63.896} C_DIS
LIN {X -0.060,Y -519.246,Z 399.152,A 0.000,B 0.000,C 90.000,E1 63.332} C_DIS
LIN {X -0.023,Y -522.380,Z 399.149,A 0.000,B 0.000,C 90.000,E1 62.743} C_DIS
LIN {X -0.115,Y -525.845,Z 399.145,A 0.000,B 0.000,C 90.000,E1 62.025} C_DIS
LIN {X 0.131,Y -527.791,Z 399.142,A 0.000,B 0.000,C 90.000,E1 61.563} C_DIS
LIN {X -0.063,Y -531.185,Z 399.137,A 0.000,B 0.000,C 90.000,E1 60.717} C_DIS
LIN {X 0.065,Y -533.219,Z 399.134,A 0.000,B 0.000,C 90.000,E1 60.127} C_DIS
LIN {X 0.210,Y -535.062,Z 399.131,A 0.000,B 0.000,C 90.000,E1 59.537} C_DIS
LIN {X 0.356,Y -537.376,Z 399.126,A 0.000,B 0.000,C 90.000,E1 58.663} C_DIS
LIN {X 0.070,Y -538.756,Z 399.123,A 0.000,B 0.000,C 90.000,E1 58.122} C_DIS
LIN {X 0.259,Y -540.475,Z 399.118,A 0.000,B 0.000,C 90.000,E1 57.248} C_DIS
LIN {X -0.008,Y -541.378,Z 399.115,A 0.000,B 0.000,C 90.000,E1 56.707} C_DIS
LIN {X -0.249,Y -542.377,Z 399.110,A 0.000,B 0.000,C 90.000,E1 55.881} C_DIS
LIN {X 0.274,Y -543.039,Z 399.106,A 0.000,B 0.000,C 90.000,E1 54.975} C_DIS
LIN {X 0.046,Y -543.333,Z 399.101,A 0.000,B 0.000,C 90.000,E1 54.149} C_DIS
LIN {X 0.137,Y -543.244,Z 399.096,A 0.000,B 0.000,C 90.000,E1 53.290} C_DIS
LIN {X -0.204,Y -542.980,Z 399.091,A 0.000,B 0.000,C 90.000,E1 52.477} C_DIS
LIN {X -0.087,Y -542.074,Z 399.085,A 0.000,B 0.000,C 90.000,E1 51.331} C_DIS
LIN {X -0.066,Y -540.955,Z 399.079,A 0.000,B 0.000,C 90.000,E1 50.194} C_DIS
LIN {X -0.055,Y -539.509,Z 399.073,A 0.000,B 0.000,C 90.000,E1 49.057} C_DIS
LIN {X -0.064,Y -537.843,Z 399.066,A 0.000,B 0.000,C 90.000,E1 47.919} C_DIS
LIN {X 0.251,Y -535.656,Z 399.058,A 0.000,B 0.000,C 90.000,E1 46.458} C_DIS
LIN {X -0.311,Y -532.730,Z 399.047,A 0.000,B 0.000,C 90.000,E1 44.514} C_DIS
LIN {X 0.190,Y -530.035,Z 399.036,A 0.000,B 0.000,C 90.000,E1 42.447} C_DIS
LIN {X -0.068,Y -527.826,Z 399.026,A 0.000,B 0.000,C 90.000,E1 40.744} C_DIS
LIN {X 0.151,Y -526.444,Z 399.020,A 0.000,B 0.000,C 90.000,E1 39.564} C_DIS
LIN {X 0.282,Y -524.265,Z 399.010,A 0.000,B 0.000,C 90.000,E1 37.810} C_DIS
LIN {X 0.090,Y -522.403,Z 399.002,A 0.000,B 0.000,C 90.000,E1 36.377} C_DIS
LIN {X -0.141,Y -520.520,Z 398.994,A 0.000,B 0.000,C 90.000,E1 34.945} C_DIS
LIN {X 0.092,Y -518.198,Z 398.984,A 0.000,B 0.000,C 90.000,E1 33.166} C_DIS
LIN {X -0.017,Y -516.617,Z 398.978,A 0.000,B 0.000,C 90.000,E1 32.005} C_DIS
LIN {X 0.210,Y -513.150,Z 398.963,A 0.000,B 0.000,C 90.000,E1 29.333} C_DIS
LIN {X -0.073,Y -510.252,Z 398.950,A 0.000,B 0.000,C 90.000,E1 27.001} C_DIS
LIN {X -0.208,Y -507.596,Z 398.937,A 0.000,B 0.000,C 90.000,E1 24.643} C_DIS
LIN {X 0.285,Y -505.266,Z 398.924,A 0.000,B 0.000,C 90.000,E1 22.206} C_DIS
LIN {X -0.146,Y -503.344,Z 398.910,A 0.000,B 0.000,C 90.000,E1 19.866} C_DIS
LIN {X -0.024,Y -501.652,Z 398.897,A 0.000,B 0.000,C 90.000,E1 17.457} C_DIS
LIN {X -0.131,Y -500.724,Z 398.889,A 0.000,B 0.000,C 90.000,E1 15.969} C_DIS
LIN {X 0.050,Y -499.322,Z 398.874,A 0.000,B 0.000,C 90.000,E1 13.244} C_DIS
LIN {X -0.126,Y -498.411,Z 398.857,A 0.000,B 0.000,C 90.000,E1 10.254} C_DIS
LIN {X 0.126,Y -498.185,Z 398.844,A 0.000,B 0.000,C 90.000,E1 7.814} C_DIS
LIN {X -0.141,Y -498.807,Z 398.825,A 0.000,B 0.000,C 90.000,E1 4.531} C_DIS
LIN {X -0.230,Y -501.077,Z 398.803,A 0.000,B 0.000,C 90.000,E1 0.630} C_DIS
LIN {X 0.177,Y -504.752,Z 398.784,A 0.000,B 0.000,C 90.000,E1 357.078} C_DIS
LIN {X -0.090,Y -508.096,Z 398.771,A 0.000,B 0.000,C 90.000,E1 354.723} C_DIS
LIN {X -0.153,Y -511.890,Z 398.757,A 0.000,B 0.000,C 90.000,E1 352.356} C_DIS
LIN {X 0.123,Y -514.582,Z 398.749,A 0.000,B 0.000,C 90.000,E1 350.849} C_DIS
LIN {X -0.105,Y -522.104,Z 398.730,A 0.000,B 0.000,C 90.000,E1 347.353} C_DIS
LIN {X 0.211,Y -527.193,Z 398.718,A 0.000,B 0.000,C 90.000,E1 345.283} C_DIS
LIN {X -0.076,Y -530.215,Z 398.712,A 0.000,B 0.000,C 90.000,E1 344.157} C_DIS
LIN {X 0.048,Y -534.786,Z 398.702,A 0.000,B 0.000,C 90.000,E1 342.417} C_DIS
LIN {X 0.231,Y -538.696,Z 398.694,A 0.000,B 0.000,C 90.000,E1 340.967} C_DIS
LIN {X -0.255,Y -544.323,Z 398.683,A 0.000,B 0.000,C 90.000,E1 339.028} C_DIS
LIN {X 0.022,Y -549.200,Z 398.674,A 0.000,B 0.000,C 90.000,E1 337.305} C_DIS
LIN {X -0.112,Y -555.005,Z 398.663,A 0.000,B 0.000,C 90.000,E1 335.357} C_DIS
LIN {X 0.142,Y -560.972,Z 398.652,A 0.000,B 0.000,C 90.000,E1 333.384} C_DIS
LIN {X 0.037,Y -567.169,Z 398.642,A 0.000,B 0.000,C 90.000,E1 331.463} C_DIS
LIN {X -0.059,Y -568.868,Z 398.638,A 0.000,B 0.000,C 90.000,E1 330.923} C_DIS
LIN {X -0.136,Y -570.754,Z 398.635,A 0.000,B 0.000,C 90.000,E1 330.383} C_DIS
LIN {X 0.086,Y -575.232,Z 398.628,A 0.000,B 0.000,C 90.000,E1 328.997} C_DIS
LIN {X 0.044,Y -578.855,Z 398.622,A 0.000,B 0.000,C 90.000,E1 327.916} C_DIS
LIN {X -0.101,Y -583.297,Z 398.614,A 0.000,B 0.000,C 90.000,E1 326.580} C_DIS
LIN {X 0.044,Y -589.618,Z 398.604,A 0.000,B 0.000,C 90.000,E1 324.689} C_DIS
LIN {X -0.130,Y -596.037,Z 398.594,A 0.000,B 0.000,C 90.000,E1 322.844} C_DIS
LIN {X -0.038,Y -601.666,Z 398.585,A 0.000,B 0.000,C 90.000,E1 321.251} C_DIS
LIN {X 0.288,Y -606.457,Z 398.577,A 0.000,B 0.000,C 90.000,E1 319.908} C_DIS
LIN {X 0.058,Y -612.115,Z 398.569,A 0.000,B 0.000,C 90.000,E1 318.366} C_DIS
LIN {X 0.273,Y -615.858,Z 398.563,A 0.000,B 0.000,C 90.000,E1 317.310} C_DIS
LIN {X -0.075,Y -620.420,Z 398.556,A 0.000,B 0.000,C 90.000,E1 316.053} C_DIS
LIN {X 0.085,Y -624.958,Z 398.549,A 0.000,B 0.000,C 90.000,E1 314.757} C_DIS
LIN {X 0.200,Y -630.557,Z 398.540,A 0.000,B 0.000,C 90.000,E1 313.218} C_DIS
LIN {X 0.031,Y -636.124,Z 398.532,A 0.000,B 0.000,C 90.000,E1 311.714} C_DIS
LIN {X 0.109,Y -639.848,Z 398.526,A 0.000,B 0.000,C 90.000,E1 310.701} C_DIS
LIN {X -0.277,Y -644.307,Z 398.519,A 0.000,B 0.000,C 90.000,E1 309.483} C_DIS
LIN {X -0.103,Y -648.551,Z 398.512,A 0.000,B 0.000,C 90.000,E1 308.222} C_DIS
LIN {X -0.187,Y -651.804,Z 398.507,A 0.000,B 0.000,C 90.000,E1 307.237} C_DIS
LIN {X 0.170,Y -656.522,Z 398.499,A 0.000,B 0.000,C 90.000,E1 305.724} C_DIS
LIN {X -0.145,Y -660.948,Z 398.490,A 0.000,B 0.000,C 90.000,E1 304.278} C_DIS
LIN {X 0.120,Y -666.071,Z 398.481,A 0.000,B 0.000,C 90.000,E1 302.546} C_DIS
LIN {X -0.371,Y -670.383,Z 398.473,A 0.000,B 0.000,C 90.000,E1 301.131} C_DIS
LIN {X 0.036,Y -673.109,Z 398.467,A 0.000,B 0.000,C 90.000,E1 300.129} C_DIS
LIN {X 0.145,Y -675.588,Z 398.462,A 0.000,B 0.000,C 90.000,E1 299.155} C_DIS
LIN {X -0.112,Y -678.415,Z 398.455,A 0.000,B 0.000,C 90.000,E1 297.975} C_DIS
LIN {X 0.070,Y -680.486,Z 398.450,A 0.000,B 0.000,C 90.000,E1 297.001} C_DIS
LIN {X 0.067,Y -681.741,Z 398.446,A 0.000,B 0.000,C 90.000,E1 296.283} C_DIS
LIN {X -0.028,Y -682.274,Z 398.445,A 0.000,B 0.000,C 90.000,E1 296.052} C_DIS
LIN {X 0.192,Y -683.786,Z 398.439,A 0.000,B 0.000,C 90.000,E1 295.079} C_DIS
LIN {X -0.081,Y -684.692,Z 398.435,A 0.000,B 0.000,C 90.000,E1 294.387} C_DIS
LIN {X 0.283,Y -685.427,Z 398.432,A 0.000,B 0.000,C 90.000,E1 293.643} C_DIS
LIN {X -0.189,Y -685.836,Z 398.429,A 0.000,B 0.000,C 90.000,E1 293.206} C_DIS
LIN {X 0.403,Y -686.105,Z 398.424,A 0.000,B 0.000,C 90.000,E1 292.206} C_DIS
LIN {X -0.109,Y -686.156,Z 398.420,A 0.000,B 0.000,C 90.000,E1 291.535} C_DIS
LIN {X 0.269,Y -686.171,Z 398.416,A 0.000,B 0.000,C 90.000,E1 290.791} C_DIS
LIN {X -0.239,Y -685.805,Z 398.412,A 0.000,B 0.000,C 90.000,E1 290.120} C_DIS
LIN {X 0.092,Y -685.090,Z 398.406,A 0.000,B 0.000,C 90.000,E1 289.141} C_DIS
LIN {X 0.220,Y -684.317,Z 398.402,A 0.000,B 0.000,C 90.000,E1 288.417} C_DIS
LIN {X 0.308,Y -683.047,Z 398.397,A 0.000,B 0.000,C 90.000,E1 287.457} C_DIS
LIN {X 0.277,Y -682.663,Z 398.396,A 0.000,B 0.000,C 90.000,E1 287.221} C_DIS
LIN {X -0.385,Y -682.199,Z 398.393,A 0.000,B 0.000,C 90.000,E1 286.804} C_DIS
LIN {X -0.221,Y -681.806,Z 398.392,A 0.000,B 0.000,C 90.000,E1 286.551} C_DIS
LIN {X -0.254,Y -681.590,Z 398.391,A 0.000,B 0.000,C 90.000,E1 286.315} C_DIS
LIN {X -0.388,Y -680.256,Z 398.385,A 0.000,B 0.000,C 90.000,E1 285.371} C_DIS
LIN {X 0.336,Y -679.163,Z 398.381,A 0.000,B 0.000,C 90.000,E1 284.592} C_DIS
LIN {X 0.037,Y -676.644,Z 398.372,A 0.000,B 0.000,C 90.000,E1 282.939} C_DIS
LIN {X 0.134,Y -673.721,Z 398.361,A 0.000,B 0.000,C 90.000,E1 281.007} C_DIS
LIN {X -0.231,Y -670.624,Z 398.348,A 0.000,B 0.000,C 90.000,E1 278.624} C_DIS
LIN {X 0.352,Y -667.849,Z 398.333,A 0.000,B 0.000,C 90.000,E1 275.910} C_DIS
LIN {X -0.164,Y -666.459,Z 398.322,A 0.000,B 0.000,C 90.000,E1 274.012} C_DIS
LIN {X -0.272,Y -665.256,Z 398.310,A 0.000,B 0.000,C 90.000,E1 271.833} C_DIS
LIN {X -0.274,Y -664.859,Z 398.305,A 0.000,B 0.000,C 90.000,E1 270.859} C_DIS
LIN {X -0.275,Y -664.240,Z 398.299,A 0.000,B 0.000,C 90.000,E1 269.885} C_DIS
LIN {X -0.289,Y -662.832,Z 398.288,A 0.000,B 0.000,C 90.000,E1 267.936} C_DIS
LIN {X -0.166,Y -661.544,Z 398.279,A 0.000,B 0.000,C 90.000,E1 266.216} C_DIS
LIN {X -0.010,Y -660.772,Z 398.275,A 0.000,B 0.000,C 90.000,E1 265.469} C_DIS
LIN {X 0.139,Y -659.671,Z 398.271,A 0.000,B 0.000,C 90.000,E1 264.723} C_DIS
LIN {X -0.185,Y -658.772,Z 398.268,A 0.000,B 0.000,C 90.000,E1 264.261} C_DIS
LIN {X 0.125,Y -655.770,Z 398.260,A 0.000,B 0.000,C 90.000,E1 262.761} C_DIS
LIN {X -0.185,Y -652.355,Z 398.252,A 0.000,B 0.000,C 90.000,E1 261.310} C_DIS
LIN {X 0.222,Y -649.187,Z 398.245,A 0.000,B 0.000,C 90.000,E1 260.038} C_DIS
LIN {X 0.040,Y -645.766,Z 398.238,A 0.000,B 0.000,C 90.000,E1 258.814} C_DIS
LIN {X -0.201,Y -642.213,Z 398.231,A 0.000,B 0.000,C 90.000,E1 257.589} C_DIS
LIN {X 0.091,Y -637.639,Z 398.223,A 0.000,B 0.000,C 90.000,E1 256.061} C_DIS
LIN {X 0.009,Y -633.598,Z 398.216,A 0.000,B 0.000,C 90.000,E1 254.810} C_DIS
LIN {X 0.072,Y -631.024,Z 398.211,A 0.000,B 0.000,C 90.000,E1 254.047} C_DIS
LIN {X 0.062,Y -626.480,Z 398.204,A 0.000,B 0.000,C 90.000,E1 252.779} C_DIS
LIN {X 0.010,Y -622.673,Z 398.199,A 0.000,B 0.000,C 90.000,E1 251.764} C_DIS
LIN {X -0.133,Y -617.824,Z 398.192,A 0.000,B 0.000,C 90.000,E1 250.496} C_DIS
LIN {X 0.104,Y -613.851,Z 398.186,A 0.000,B 0.000,C 90.000,E1 249.444} C_DIS
LIN {X 0.027,Y -608.623,Z 398.179,A 0.000,B 0.000,C 90.000,E1 248.156} C_DIS
LIN {X -0.148,Y -603.215,Z 398.171,A 0.000,B 0.000,C 90.000,E1 246.869} C_DIS
LIN {X 0.058,Y -597.687,Z 398.164,A 0.000,B 0.000,C 90.000,E1 245.537} C_DIS
LIN {X 0.083,Y -590.998,Z 398.155,A 0.000,B 0.000,C 90.000,E1 243.948} C_DIS
LIN {X -0.035,Y -584.264,Z 398.146,A 0.000,B 0.000,C 90.000,E1 242.359} C_DIS
LIN {X 0.246,Y -577.670,Z 398.138,A 0.000,B 0.000,C 90.000,E1 240.717} C_DIS
LIN {X 0.151,Y -568.088,Z 398.124,A 0.000,B 0.000,C 90.000,E1 238.280} C_DIS
LIN {X 0.172,Y -559.136,Z 398.110,A 0.000,B 0.000,C 90.000,E1 235.801} C_DIS
LIN {X 0.026,Y -553.432,Z 398.101,A 0.000,B 0.000,C 90.000,E1 234.149} C_DIS
LIN {X -0.038,Y -547.773,Z 398.092,A 0.000,B 0.000,C 90.000,E1 232.477} C_DIS
LIN {X -0.246,Y -542.940,Z 398.084,A 0.000,B 0.000,C 90.000,E1 231.090} C_DIS
LIN {X 0.216,Y -538.190,Z 398.076,A 0.000,B 0.000,C 90.000,E1 229.622} C_DIS
LIN {X -0.311,Y -530.868,Z 398.063,A 0.000,B 0.000,C 90.000,E1 227.391} C_DIS
LIN {X -0.199,Y -525.576,Z 398.054,A 0.000,B 0.000,C 90.000,E1 225.648} C_DIS
LIN {X -0.283,Y -519.438,Z 398.042,A 0.000,B 0.000,C 90.000,E1 223.623} C_DIS
LIN {X 0.218,Y -513.462,Z 398.031,A 0.000,B 0.000,C 90.000,E1 221.515} C_DIS
LIN {X -0.213,Y -506.893,Z 398.018,A 0.000,B 0.000,C 90.000,E1 219.197} C_DIS
LIN {X 0.071,Y -501.419,Z 398.006,A 0.000,B 0.000,C 90.000,E1 217.076} C_DIS
LIN {X -0.259,Y -496.848,Z 397.996,A 0.000,B 0.000,C 90.000,E1 215.311} C_DIS
LIN {X -0.020,Y -491.698,Z 397.984,A 0.000,B 0.000,C 90.000,E1 213.166} C_DIS
LIN {X -0.015,Y -487.437,Z 397.974,A 0.000,B 0.000,C 90.000,E1 211.337} C_DIS
LIN {X -0.137,Y -482.506,Z 397.962,A 0.000,B 0.000,C 90.000,E1 209.205} C_DIS
LIN {X 0.016,Y -478.204,Z 397.952,A 0.000,B 0.000,C 90.000,E1 207.334} C_DIS
LIN {X -0.076,Y -475.278,Z 397.945,A 0.000,B 0.000,C 90.000,E1 206.104} C_DIS
LIN {X 0.126,Y -470.748,Z 397.935,A 0.000,B 0.000,C 90.000,E1 204.207} C_DIS
LIN {X 0.085,Y -466.929,Z 397.926,A 0.000,B 0.000,C 90.000,E1 202.642} C_DIS
LIN {X 0.156,Y -462.404,Z 397.915,A 0.000,B 0.000,C 90.000,E1 200.737} C_DIS
LIN {X 0.221,Y -456.723,Z 397.901,A 0.000,B 0.000,C 90.000,E1 198.181} C_DIS
LIN {X -0.174,Y -451.468,Z 397.887,A 0.000,B 0.000,C 90.000,E1 195.662} C_DIS
LIN {X -0.096,Y -446.725,Z 397.873,A 0.000,B 0.000,C 90.000,E1 193.063} C_DIS
LIN {X 0.009,Y -443.917,Z 397.864,A 0.000,B 0.000,C 90.000,E1 191.422} C_DIS
LIN {X -0.024,Y -441.275,Z 397.854,A 0.000,B 0.000,C 90.000,E1 189.792} C_DIS
LIN {X 0.124,Y -437.857,Z 397.842,A 0.000,B 0.000,C 90.000,E1 187.473} C_DIS
LIN {X 0.088,Y -433.211,Z 397.821,A 0.000,B 0.000,C 90.000,E1 183.841} C_DIS
LIN {X -0.009,Y -430.241,Z 397.805,A 0.000,B 0.000,C 90.000,E1 180.859} C_DIS
LIN {X 0.133,Y -427.495,Z 397.779,A 0.000,B 0.000,C 90.000,E1 176.159} C_DIS
LIN {X -0.052,Y -426.808,Z 397.762,A 0.000,B 0.000,C 90.000,E1 173.166} C_DIS
LIN {X -0.057,Y -427.977,Z 397.730,A 0.000,B 0.000,C 90.000,E1 167.465} C_DIS
LIN {X 0.206,Y -431.765,Z 397.703,A 0.000,B 0.000,C 90.000,E1 162.417} C_DIS
LIN {X 0.199,Y -436.844,Z 397.679,A 0.000,B 0.000,C 90.000,E1 158.103} C_DIS
LIN {X 0.208,Y -442.986,Z 397.657,A 0.000,B 0.000,C 90.000,E1 154.152} C_DIS
LIN {X 0.040,Y -449.901,Z 397.637,A 0.000,B 0.000,C 90.000,E1 150.589} C_DIS
LIN {X -0.037,Y -457.426,Z 397.619,A 0.000,B 0.000,C 90.000,E1 147.375} C_DIS
LIN {X 0.047,Y -467.128,Z 397.599,A 0.000,B 0.000,C 90.000,E1 143.863} C_DIS
LIN {X -0.171,Y -475.005,Z 397.585,A 0.000,B 0.000,C 90.000,E1 141.376} C_DIS
LIN {X -0.236,Y -480.115,Z 397.577,A 0.000,B 0.000,C 90.000,E1 139.828} C_DIS
LIN {X -0.027,Y -484.193,Z 397.570,A 0.000,B 0.000,C 90.000,E1 138.566} C_DIS
LIN {X 0.057,Y -487.236,Z 397.565,A 0.000,B 0.000,C 90.000,E1 137.634} C_DIS
LIN {X -0.018,Y -490.977,Z 397.558,A 0.000,B 0.000,C 90.000,E1 136.419} C_DIS
LIN {X -0.025,Y -494.522,Z 397.551,A 0.000,B 0.000,C 90.000,E1 135.202} C_DIS
LIN {X -0.340,Y -497.748,Z 397.544,A 0.000,B 0.000,C 90.000,E1 134.028} C_DIS
LIN {X -0.097,Y -499.973,Z 397.539,A 0.000,B 0.000,C 90.000,E1 133.095} C_DIS
LIN {X 0.176,Y -501.953,Z 397.534,A 0.000,B 0.000,C 90.000,E1 132.162} C_DIS
LIN {X -0.027,Y -504.122,Z 397.528,A 0.000,B 0.000,C 90.000,E1 130.987} C_DIS
LIN {X -0.043,Y -505.491,Z 397.523,A 0.000,B 0.000,C 90.000,E1 130.092} C_DIS
LIN {X -0.040,Y -506.510,Z 397.518,A 0.000,B 0.000,C 90.000,E1 129.197} C_DIS
LIN {X 0.071,Y -506.963,Z 397.514,A 0.000,B 0.000,C 90.000,E1 128.588} C_DIS
LIN {X -0.130,Y -507.218,Z 397.511,A 0.000,B 0.000,C 90.000,E1 128.016} C_DIS
LIN {X 0.075,Y -507.131,Z 397.508,A 0.000,B 0.000,C 90.000,E1 127.397} C_DIS
LIN {X 0.187,Y -506.817,Z 397.505,A 0.000,B 0.000,C 90.000,E1 126.790} C_DIS
LIN {X -0.114,Y -505.969,Z 397.500,A 0.000,B 0.000,C 90.000,E1 125.931} C_DIS
LIN {X 0.092,Y -505.194,Z 397.496,A 0.000,B 0.000,C 90.000,E1 125.311} C_DIS
LIN {X 0.076,Y -503.179,Z 397.490,A 0.000,B 0.000,C 90.000,E1 124.119} C_DIS
LIN {X -0.038,Y -502.656,Z 397.488,A 0.000,B 0.000,C 90.000,E1 123.833} C_DIS
LIN {X -0.252,Y -500.499,Z 397.483,A 0.000,B 0.000,C 90.000,E1 122.959} C_DIS
LIN {X 0.068,Y -496.932,Z 397.476,A 0.000,B 0.000,C 90.000,E1 121.720} C_DIS
LIN {X 0.220,Y -493.839,Z 397.471,A 0.000,B 0.000,C 90.000,E1 120.797} C_DIS
LIN {X -0.075,Y -489.225,Z 397.465,A 0.000,B 0.000,C 90.000,E1 119.617} C_DIS
LIN {X -0.009,Y -485.354,Z 397.459,A 0.000,B 0.000,C 90.000,E1 118.693} C_DIS
LIN {X -0.213,Y -480.623,Z 397.453,A 0.000,B 0.000,C 90.000,E1 117.641} C_DIS
LIN {X -0.090,Y -474.049,Z 397.446,A 0.000,B 0.000,C 90.000,E1 116.232} C_DIS
LIN {X 0.002,Y -469.508,Z 397.441,A 0.000,B 0.000,C 90.000,E1 115.283} C_DIS
LIN {X -0.265,Y -462.541,Z 397.433,A 0.000,B 0.000,C 90.000,E1 113.898} C_DIS
LIN {X -0.137,Y -457.112,Z 397.426,A 0.000,B 0.000,C 90.000,E1 112.770} C_DIS
LIN {X 0.034,Y -452.104,Z 397.421,A 0.000,B 0.000,C 90.000,E1 111.716} C_DIS
LIN {X -0.006,Y -452.117,Z 397.421,A 0.000,B 0.000,C 90.000,E1 111.716} C_DIS
LIN {X -0.044,Y -457.122,Z 397.410,A 0.000,B 0.000,C 90.000,E1 109.866} C_DIS
LIN {X -0.195,Y -466.520,Z 397.386,A 0.000,B 0.000,C 90.000,E1 105.426} C_DIS
LIN {X -0.020,Y -467.983,Z 397.382,A 0.000,B 0.000,C 90.000,E1 104.773} C_DIS
LIN {X -0.057,Y -476.201,Z 397.356,A 0.000,B 0.000,C 90.000,E1 100.074} C_DIS
LIN {X 0.199,Y -482.104,Z 397.330,A 0.000,B 0.000,C 90.000,E1 95.391} C_DIS
LIN {X -0.052,Y -485.515,Z 397.304,A 0.000,B 0.000,C 90.000,E1 90.802} C_DIS
LIN {X -0.019,Y -486.382,Z 397.281,A 0.000,B 0.000,C 90.000,E1 86.502} C_DIS
LIN {X -0.195,Y -486.359,Z 397.279,A 0.000,B 0.000,C 90.000,E1 86.216} C_DIS
LIN {X -0.111,Y -484.680,Z 397.253,A 0.000,B 0.000,C 90.000,E1 81.602} C_DIS
LIN {X 0.257,Y -480.598,Z 397.228,A 0.000,B 0.000,C 90.000,E1 76.937} C_DIS
LIN {X 0.115,Y -480.219,Z 397.226,A 0.000,B 0.000,C 90.000,E1 76.645} C_DIS
LIN {X 0.004,Y -474.050,Z 397.200,A 0.000,B 0.000,C 90.000,E1 72.000} C_DIS
LIN {X -0.238,Y -471.137,Z 397.192,A 0.000,B 0.000,C 90.000,E1 70.550} C_DIS
LIN {X 0.165,Y -471.168,Z 397.192,A 0.000,B 0.000,C 90.000,E1 70.496} C_DIS
LIN {X -0.161,Y -481.043,Z 397.184,A 0.000,B 0.000,C 90.000,E1 69.209} C_DIS
LIN {X -0.141,Y -490.168,Z 397.178,A 0.000,B 0.000,C 90.000,E1 67.975} C_DIS
LIN {X -0.239,Y -497.971,Z 397.172,A 0.000,B 0.000,C 90.000,E1 66.922} C_DIS
LIN {X 0.157,Y -504.261,Z 397.167,A 0.000,B 0.000,C 90.000,E1 65.973} C_DIS
LIN {X -0.135,Y -508.295,Z 397.163,A 0.000,B 0.000,C 90.000,E1 65.409} C_DIS
LIN {X -0.296,Y -513.798,Z 397.158,A 0.000,B 0.000,C 90.000,E1 64.537} C_DIS
LIN {X 0.161,Y -517.154,Z 397.155,A 0.000,B 0.000,C 90.000,E1 63.896} C_DIS
LIN {X -0.179,Y -518.641,Z 397.154,A 0.000,B 0.000,C 90.000,E1 63.640} C_DIS
LIN {X -0.049,Y -520.292,Z 397.152,A 0.000,B 0.000,C 90.000,E1 63.332} C_DIS
LIN {X -0.003,Y -523.278,Z 397.149,A 0.000,B 0.000,C 90.000,E1 62.743} C_DIS
LIN {X 0.069,Y -526.025,Z 397.145,A 0.000,B 0.000,C 90.000,E1 62.153} C_DIS
LIN {X 0.066,Y -527.818,Z 397.143,A 0.000,B 0.000,C 90.000,E1 61.719} C_DIS
LIN {X 0.010,Y -529.052,Z 397.141,A 0.000,B 0.000,C 90.000,E1 61.435} C_DIS
LIN {X 0.126,Y -531.271,Z 397.138,A 0.000,B 0.000,C 90.000,E1 60.845} C_DIS
LIN {X -0.036,Y -534.159,Z 397.133,A 0.000,B 0.000,C 90.000,E1 59.999} C_DIS
LIN {X 0.113,Y -535.947,Z 397.130,A 0.000,B 0.000,C 90.000,E1 59.410} C_DIS
LIN {X 0.268,Y -538.188,Z 397.125,A 0.000,B 0.000,C 90.000,E1 58.535} C_DIS
LIN {X -0.006,Y -540.129,Z 397.121,A 0.000,B 0.000,C 90.000,E1 57.709} C_DIS
LIN {X -0.286,Y -540.727,Z 397.119,A 0.000,B 0.000,C 90.000,E1 57.454} C_DIS
LIN {X -0.081,Y -542.089,Z 397.114,A 0.000,B 0.000,C 90.000,E1 56.580} C_DIS
LIN {X -0.012,Y -543.046,Z 397.110,A 0.000,B 0.000,C 90.000,E1 55.722} C_DIS
LIN {X -0.233,Y -543.806,Z 397.105,A 0.000,B 0.000,C 90.000,E1 54.895} C_DIS
LIN {X -0.133,Y -544.131,Z 397.100,A 0.000,B 0.000,C 90.000,E1 54.036} C_DIS
LIN {X 0.011,Y -543.975,Z 397.094,A 0.000,B 0.000,C 90.000,E1 52.889} C_DIS
LIN {X 0.081,Y -543.832,Z 397.091,A 0.000,B 0.000,C 90.000,E1 52.316} C_DIS
LIN {X 0.213,Y -542.999,Z 397.084,A 0.000,B 0.000,C 90.000,E1 51.170} C_DIS
LIN {X -0.098,Y -541.815,Z 397.078,A 0.000,B 0.000,C 90.000,E1 50.070} C_DIS
LIN {X -0.079,Y -540.362,Z 397.072,A 0.000,B 0.000,C 90.000,E1 48.933} C_DIS
LIN {X 0.283,Y -538.313,Z 397.064,A 0.000,B 0.000,C 90.000,E1 47.472} C_DIS
LIN {X -0.233,Y -534.817,Z 397.051,A 0.000,B 0.000,C 90.000,E1 45.243} C_DIS
LIN {X -0.061,Y -532.028,Z 397.040,A 0.000,B 0.000,C 90.000,E1 43.218} C_DIS
LIN {X -0.300,Y -529.434,Z 397.029,A 0.000,B 0.000,C 90.000,E1 41.229} C_DIS
LIN {X -0.171,Y -527.287,Z 397.019,A 0.000,B 0.000,C 90.000,E1 39.483} C_DIS
LIN {X -0.023,Y -525.105,Z 397.010,A 0.000,B 0.000,C 90.000,E1 37.729} C_DIS
LIN {X -0.163,Y -523.627,Z 397.003,A 0.000,B 0.000,C 90.000,E1 36.583} C_DIS
LIN {X 0.008,Y -521.332,Z 396.993,A 0.000,B 0.000,C 90.000,E1 34.818} C_DIS
LIN {X -0.170,Y -519.029,Z 396.984,A 0.000,B 0.000,C 90.000,E1 33.086} C_DIS
LIN {X 0.169,Y -517.422,Z 396.977,A 0.000,B 0.000,C 90.000,E1 31.878} C_DIS
LIN {X -0.274,Y -514.023,Z 396.963,A 0.000,B 0.000,C 90.000,E1 29.283} C_DIS
LIN {X 0.168,Y -511.109,Z 396.949,A 0.000,B 0.000,C 90.000,E1 26.873} C_DIS
LIN {X -0.044,Y -508.820,Z 396.938,A 0.000,B 0.000,C 90.000,E1 24.823} C_DIS
LIN {X -0.085,Y -506.205,Z 396.923,A 0.000,B 0.000,C 90.000,E1 22.153} C_DIS
LIN {X 0.078,Y -504.053,Z 396.908,A 0.000,B 0.000,C 90.000,E1 19.450} C_DIS
LIN {X 0.157,Y -502.600,Z 396.897,A 0.000,B 0.000,C 90.000,E1 17.347} C_DIS
LIN {X 0.213,Y -501.712,Z 396.888,A 0.000,B 0.000,C 90.000,E1 15.843} C_DIS
LIN {X -0.072,Y -500.343,Z 396.873,A 0.000,B 0.000,C 90.000,E1 13.175} C_DIS
LIN {X 0.099,Y -499.456,Z 396.855,A 0.000,B 0.000,C 90.000,E1 9.849} C_DIS
LIN {X -0.112,Y -499.346,Z 396.841,A 0.000,B 0.000,C 90.000,E1 7.466} C_DIS
LIN {X -0.113,Y -499.930,Z 396.826,A 0.000,B 0.000,C 90.000,E1 4.759} C_DIS
LIN {X -0.154,Y -502.153,Z 396.805,A 0.000,B 0.000,C 90.000,E1 0.859} C_DIS
LIN {X 0.221,Y -506.066,Z 396.784,A 0.000,B 0.000,C 90.000,E1 357.078} C_DIS
LIN {X -0.008,Y -509.409,Z 396.771,A 0.000,B 0.000,C 90.000,E1 354.723} C_DIS
LIN {X -0.032,Y -513.232,Z 396.758,A 0.000,B 0.000,C 90.000,E1 352.356} C_DIS
LIN {X 0.149,Y -517.110,Z 396.746,A 0.000,B 0.000,C 90.000,E1 350.274} C_DIS
LIN {X 0.095,Y -522.126,Z 396.733,A 0.000,B 0.000,C 90.000,E1 347.937} C_DIS
LIN {X -0.222,Y -527.128,Z 396.722,A 0.000,B 0.000,C 90.000,E1 345.936} C_DIS
LIN {X 0.195,Y -531.662,Z 396.712,A 0.000,B 0.000,C 90.000,E1 344.157} C_DIS
LIN {X 0.156,Y -535.493,Z 396.704,A 0.000,B 0.000,C 90.000,E1 342.725} C_DIS
LIN {X -0.163,Y -539.440,Z 396.696,A 0.000,B 0.000,C 90.000,E1 341.329} C_DIS
LIN {X -0.123,Y -545.040,Z 396.685,A 0.000,B 0.000,C 90.000,E1 339.337} C_DIS
LIN {X -0.072,Y -550.695,Z 396.674,A 0.000,B 0.000,C 90.000,E1 337.358} C_DIS
LIN {X 0.059,Y -555.687,Z 396.665,A 0.000,B 0.000,C 90.000,E1 335.665} C_DIS
LIN {X 0.088,Y -561.622,Z 396.654,A 0.000,B 0.000,C 90.000,E1 333.717} C_DIS
LIN {X 0.079,Y -568.662,Z 396.642,A 0.000,B 0.000,C 90.000,E1 331.513} C_DIS
LIN {X -0.002,Y -570.335,Z 396.639,A 0.000,B 0.000,C 90.000,E1 330.973} C_DIS
LIN {X 0.147,Y -572.270,Z 396.636,A 0.000,B 0.000,C 90.000,E1 330.411} C_DIS
LIN {X 0.030,Y -577.628,Z 396.627,A 0.000,B 0.000,C 90.000,E1 328.791} C_DIS
LIN {X 0.023,Y -581.233,Z 396.621,A 0.000,B 0.000,C 90.000,E1 327.709} C_DIS
LIN {X 0.100,Y -586.598,Z 396.612,A 0.000,B 0.000,C 90.000,E1 326.087} C_DIS
LIN {X -0.081,Y -591.144,Z 396.604,A 0.000,B 0.000,C 90.000,E1 324.769} C_DIS
LIN {X -0.094,Y -596.651,Z 396.595,A 0.000,B 0.000,C 90.000,E1 323.176} C_DIS
LIN {X -0.352,Y -602.309,Z 396.587,A 0.000,B 0.000,C 90.000,E1 321.618} C_DIS
LIN {X 0.247,Y -608.021,Z 396.578,A 0.000,B 0.000,C 90.000,E1 319.989} C_DIS
LIN {X 0.046,Y -613.671,Z 396.569,A 0.000,B 0.000,C 90.000,E1 318.447} C_DIS
LIN {X 0.283,Y -617.441,Z 396.563,A 0.000,B 0.000,C 90.000,E1 317.391} C_DIS
LIN {X -0.039,Y -622.002,Z 396.556,A 0.000,B 0.000,C 90.000,E1 316.134} C_DIS
LIN {X 0.281,Y -625.701,Z 396.551,A 0.000,B 0.000,C 90.000,E1 315.081} C_DIS
LIN {X -0.250,Y -633.067,Z 396.539,A 0.000,B 0.000,C 90.000,E1 313.095} C_DIS
LIN {X 0.063,Y -638.651,Z 396.531,A 0.000,B 0.000,C 90.000,E1 311.553} C_DIS
LIN {X 0.263,Y -641.440,Z 396.527,A 0.000,B 0.000,C 90.000,E1 310.782} C_DIS
LIN {X -0.095,Y -645.887,Z 396.520,A 0.000,B 0.000,C 90.000,E1 309.564} C_DIS
LIN {X 0.109,Y -650.155,Z 396.513,A 0.000,B 0.000,C 90.000,E1 308.302} C_DIS
LIN {X -0.020,Y -654.215,Z 396.506,A 0.000,B 0.000,C 90.000,E1 307.076} C_DIS
LIN {X -0.088,Y -658.136,Z 396.499,A 0.000,B 0.000,C 90.000,E1 305.851} C_DIS
LIN {X -0.380,Y -662.571,Z 396.491,A 0.000,B 0.000,C 90.000,E1 304.405} C_DIS
LIN {X -0.083,Y -667.724,Z 396.482,A 0.000,B 0.000,C 90.000,E1 302.673} C_DIS
LIN {X 0.027,Y -672.065,Z 396.473,A 0.000,B 0.000,C 90.000,E1 301.209} C_DIS
LIN {X -0.120,Y -674.726,Z 396.468,A 0.000,B 0.000,C 90.000,E1 300.256} C_DIS
LIN {X 0.195,Y -677.761,Z 396.461,A 0.000,B 0.000,C 90.000,E1 299.027} C_DIS
LIN {X -0.227,Y -679.999,Z 396.456,A 0.000,B 0.000,C 90.000,E1 298.103} C_DIS
LIN {X -0.024,Y -682.077,Z 396.451,A 0.000,B 0.000,C 90.000,E1 297.129} C_DIS
LIN {X 0.110,Y -684.122,Z 396.444,A 0.000,B 0.000,C 90.000,E1 295.924} C_DIS
LIN {X 0.064,Y -685.398,Z 396.439,A 0.000,B 0.000,C 90.000,E1 294.975} C_DIS
LIN {X -0.122,Y -685.953,Z 396.436,A 0.000,B 0.000,C 90.000,E1 294.515} C_DIS
LIN {X 0.254,Y -686.555,Z 396.432,A 0.000,B 0.000,C 90.000,E1 293.770} C_DIS
LIN {X -0.211,Y -686.886,Z 396.430,A 0.000,B 0.000,C 90.000,E1 293.334} C_DIS
LIN {X -0.282,Y -686.988,Z 396.423,A 0.000,B 0.000,C 90.000,E1 292.153} C_DIS
LIN {X 0.282,Y -686.678,Z 396.416,A 0.000,B 0.000,C 90.000,E1 290.918} C_DIS
LIN {X -0.049,Y -685.842,Z 396.410,A 0.000,B 0.000,C 90.000,E1 289.758} C_DIS
LIN {X 0.282,Y -685.007,Z 396.405,A 0.000,B 0.000,C 90.000,E1 288.779} C_DIS
LIN {X 0.223,Y -684.406,Z 396.402,A 0.000,B 0.000,C 90.000,E1 288.308} C_DIS
LIN {X -0.331,Y -683.059,Z 396.397,A 0.000,B 0.000,C 90.000,E1 287.402} C_DIS
LIN {X -0.167,Y -680.524,Z 396.387,A 0.000,B 0.000,C 90.000,E1 285.717} C_DIS
LIN {X -0.314,Y -678.986,Z 396.382,A 0.000,B 0.000,C 90.000,E1 284.773} C_DIS
LIN {X 0.001,Y -675.867,Z 396.371,A 0.000,B 0.000,C 90.000,E1 282.827} C_DIS
LIN {X 0.146,Y -673.225,Z 396.362,A 0.000,B 0.000,C 90.000,E1 281.130} C_DIS
LIN {X -0.219,Y -670.024,Z 396.349,A 0.000,B 0.000,C 90.000,E1 278.746} C_DIS
LIN {X -0.298,Y -667.203,Z 396.334,A 0.000,B 0.000,C 90.000,E1 276.087} C_DIS
LIN {X -0.149,Y -665.825,Z 396.323,A 0.000,B 0.000,C 90.000,E1 274.131} C_DIS
LIN {X 0.265,Y -664.583,Z 396.309,A 0.000,B 0.000,C 90.000,E1 271.661} C_DIS
LIN {X 0.256,Y -664.297,Z 396.304,A 0.000,B 0.000,C 90.000,E1 270.688} C_DIS
LIN {X 0.248,Y -663.731,Z 396.299,A 0.000,B 0.000,C 90.000,E1 269.714} C_DIS
LIN {X -0.266,Y -662.953,Z 396.289,A 0.000,B 0.000,C 90.000,E1 268.051} C_DIS
LIN {X 0.220,Y -662.225,Z 396.282,A 0.000,B 0.000,C 90.000,E1 266.788} C_DIS
LIN {X 0.208,Y -661.433,Z 396.277,A 0.000,B 0.000,C 90.000,E1 265.812} C_DIS
LIN {X -0.159,Y -660.846,Z 396.274,A 0.000,B 0.000,C 90.000,E1 265.355} C_DIS
LIN {X -0.011,Y -659.768,Z 396.270,A 0.000,B 0.000,C 90.000,E1 264.609} C_DIS
LIN {X 0.193,Y -658.443,Z 396.266,A 0.000,B 0.000,C 90.000,E1 263.856} C_DIS
LIN {X -0.007,Y -657.925,Z 396.265,A 0.000,B 0.000,C 90.000,E1 263.628} C_DIS
LIN {X -0.339,Y -657.209,Z 396.262,A 0.000,B 0.000,C 90.000,E1 263.166} C_DIS
LIN {X -0.152,Y -655.723,Z 396.258,A 0.000,B 0.000,C 90.000,E1 262.413} C_DIS
LIN {X -0.198,Y -653.600,Z 396.252,A 0.000,B 0.000,C 90.000,E1 261.432} C_DIS
LIN {X 0.332,Y -650.635,Z 396.245,A 0.000,B 0.000,C 90.000,E1 260.151} C_DIS
LIN {X 0.178,Y -647.337,Z 396.239,A 0.000,B 0.000,C 90.000,E1 258.926} C_DIS
LIN {X 0.260,Y -645.294,Z 396.234,A 0.000,B 0.000,C 90.000,E1 258.173} C_DIS
LIN {X 0.299,Y -642.445,Z 396.229,A 0.000,B 0.000,C 90.000,E1 257.173} C_DIS
LIN {X 0.140,Y -638.651,Z 396.222,A 0.000,B 0.000,C 90.000,E1 255.936} C_DIS
LIN {X -0.086,Y -634.635,Z 396.215,A 0.000,B 0.000,C 90.000,E1 254.700} C_DIS
LIN {X 0.158,Y -632.073,Z 396.211,A 0.000,B 0.000,C 90.000,E1 253.921} C_DIS
LIN {X -0.016,Y -627.552,Z 396.204,A 0.000,B 0.000,C 90.000,E1 252.670} C_DIS
LIN {X 0.154,Y -624.711,Z 396.200,A 0.000,B 0.000,C 90.000,E1 251.891} C_DIS
LIN {X 0.244,Y -619.877,Z 396.192,A 0.000,B 0.000,C 90.000,E1 250.604} C_DIS
LIN {X 0.051,Y -614.898,Z 396.185,A 0.000,B 0.000,C 90.000,E1 249.337} C_DIS
LIN {X 0.209,Y -609.674,Z 396.178,A 0.000,B 0.000,C 90.000,E1 248.028} C_DIS
LIN {X 0.051,Y -604.222,Z 396.171,A 0.000,B 0.000,C 90.000,E1 246.741} C_DIS
LIN {X 0.275,Y -598.705,Z 396.164,A 0.000,B 0.000,C 90.000,E1 245.409} C_DIS
LIN {X 0.059,Y -592.015,Z 396.155,A 0.000,B 0.000,C 90.000,E1 243.845} C_DIS
LIN {X 0.219,Y -585.293,Z 396.146,A 0.000,B 0.000,C 90.000,E1 242.231} C_DIS
LIN {X -0.132,Y -579.802,Z 396.138,A 0.000,B 0.000,C 90.000,E1 240.923} C_DIS
LIN {X -0.038,Y -569.170,Z 396.123,A 0.000,B 0.000,C 90.000,E1 238.201} C_DIS
LIN {X -0.070,Y -561.219,Z 396.111,A 0.000,B 0.000,C 90.000,E1 236.008} C_DIS
LIN {X 0.157,Y -555.541,Z 396.102,A 0.000,B 0.000,C 90.000,E1 234.322} C_DIS
LIN {X -0.183,Y -549.893,Z 396.093,A 0.000,B 0.000,C 90.000,E1 232.683} C_DIS
LIN {X 0.033,Y -546.081,Z 396.086,A 0.000,B 0.000,C 90.000,E1 231.537} C_DIS
LIN {X 0.180,Y -539.367,Z 396.075,A 0.000,B 0.000,C 90.000,E1 229.542} C_DIS
LIN {X -0.313,Y -532.040,Z 396.063,A 0.000,B 0.000,C 90.000,E1 227.310} C_DIS
LIN {X -0.175,Y -526.738,Z 396.053,A 0.000,B 0.000,C 90.000,E1 225.567} C_DIS
LIN {X 0.063,Y -519.754,Z 396.040,A 0.000,B 0.000,C 90.000,E1 223.218} C_DIS
LIN {X -0.040,Y -514.605,Z 396.030,A 0.000,B 0.000,C 90.000,E1 221.472} C_DIS
LIN {X -0.011,Y -508.821,Z 396.019,A 0.000,B 0.000,C 90.000,E1 219.402} C_DIS
LIN {X 0.118,Y -504.087,Z 396.009,A 0.000,B 0.000,C 90.000,E1 217.604} C_DIS
LIN {X 0.146,Y -499.512,Z 395.999,A 0.000,B 0.000,C 90.000,E1 215.804} C_DIS
LIN {X -0.103,Y -493.557,Z 395.986,A 0.000,B 0.000,C 90.000,E1 213.420} C_DIS
LIN {X -0.154,Y -490.697,Z 395.979,A 0.000,B 0.000,C 90.000,E1 212.212} C_DIS
LIN {X 0.243,Y -486.427,Z 395.969,A 0.000,B 0.000,C 90.000,E1 210.335} C_DIS
LIN {X -0.152,Y -483.642,Z 395.962,A 0.000,B 0.000,C 90.000,E1 209.155} C_DIS
LIN {X 0.255,Y -479.359,Z 395.952,A 0.000,B 0.000,C 90.000,E1 207.257} C_DIS
LIN {X 0.149,Y -475.653,Z 395.943,A 0.000,B 0.000,C 90.000,E1 205.720} C_DIS
LIN {X -0.267,Y -471.184,Z 395.933,A 0.000,B 0.000,C 90.000,E1 203.898} C_DIS
LIN {X 0.032,Y -465.843,Z 395.920,A 0.000,B 0.000,C 90.000,E1 201.663} C_DIS
LIN {X 0.280,Y -459.297,Z 395.905,A 0.000,B 0.000,C 90.000,E1 198.779} C_DIS
LIN {X 0.038,Y -452.634,Z 395.887,A 0.000,B 0.000,C 90.000,E1 195.607} C_DIS
LIN {X 0.156,Y -447.867,Z 395.872,A 0.000,B 0.000,C 90.000,E1 193.008} C_DIS
LIN {X -0.238,Y -443.962,Z 395.860,A 0.000,B 0.000,C 90.000,E1 190.782} C_DIS
LIN {X 0.167,Y -441.367,Z 395.851,A 0.000,B 0.000,C 90.000,E1 189.095} C_DIS
LIN {X 0.165,Y -438.451,Z 395.840,A 0.000,B 0.000,C 90.000,E1 187.125} C_DIS
LIN {X 0.028,Y -434.257,Z 395.821,A 0.000,B 0.000,C 90.000,E1 183.841} C_DIS
LIN {X -0.032,Y -431.241,Z 395.805,A 0.000,B 0.000,C 90.000,E1 180.859} C_DIS
LIN {X 0.102,Y -428.604,Z 395.781,A 0.000,B 0.000,C 90.000,E1 176.502} C_DIS
LIN {X 0.015,Y -427.751,Z 395.762,A 0.000,B 0.000,C 90.000,E1 173.166} C_DIS
LIN {X 0.101,Y -428.439,Z 395.736,A 0.000,B 0.000,C 90.000,E1 168.465} C_DIS
LIN {X 0.142,Y -430.323,Z 395.717,A 0.000,B 0.000,C 90.000,E1 165.117} C_DIS
LIN {X -0.112,Y -433.325,Z 395.699,A 0.000,B 0.000,C 90.000,E1 161.819} C_DIS
LIN {X 0.028,Y -437.741,Z 395.679,A 0.000,B 0.000,C 90.000,E1 158.156} C_DIS
LIN {X 0.090,Y -443.922,Z 395.657,A 0.000,B 0.000,C 90.000,E1 154.204} C_DIS
LIN {X -0.080,Y -452.275,Z 395.633,A 0.000,B 0.000,C 90.000,E1 149.999} C_DIS
LIN {X -0.074,Y -460.047,Z 395.615,A 0.000,B 0.000,C 90.000,E1 146.786} C_DIS
LIN {X -0.146,Y -469.128,Z 395.598,A 0.000,B 0.000,C 90.000,E1 143.623} C_DIS
LIN {X -0.008,Y -476.095,Z 395.586,A 0.000,B 0.000,C 90.000,E1 141.412} C_DIS
LIN {X 0.139,Y -480.203,Z 395.579,A 0.000,B 0.000,C 90.000,E1 140.150} C_DIS
LIN {X -0.016,Y -484.308,Z 395.572,A 0.000,B 0.000,C 90.000,E1 138.933} C_DIS
LIN {X -0.109,Y -488.394,Z 395.565,A 0.000,B 0.000,C 90.000,E1 137.715} C_DIS
LIN {X 0.187,Y -492.147,Z 395.558,A 0.000,B 0.000,C 90.000,E1 136.458} C_DIS
LIN {X 0.190,Y -495.681,Z 395.552,A 0.000,B 0.000,C 90.000,E1 135.243} C_DIS
LIN {X 0.248,Y -498.998,Z 395.545,A 0.000,B 0.000,C 90.000,E1 134.028} C_DIS
LIN {X 0.142,Y -501.207,Z 395.540,A 0.000,B 0.000,C 90.000,E1 133.137} C_DIS
LIN {X 0.086,Y -503.193,Z 395.535,A 0.000,B 0.000,C 90.000,E1 132.243} C_DIS
LIN {X -0.098,Y -505.378,Z 395.528,A 0.000,B 0.000,C 90.000,E1 131.067} C_DIS
LIN {X 0.009,Y -506.390,Z 395.525,A 0.000,B 0.000,C 90.000,E1 130.458} C_DIS
LIN {X 0.020,Y -507.598,Z 395.520,A 0.000,B 0.000,C 90.000,E1 129.564} C_DIS
LIN {X 0.043,Y -508.407,Z 395.515,A 0.000,B 0.000,C 90.000,E1 128.669} C_DIS
LIN {X -0.242,Y -508.762,Z 395.510,A 0.000,B 0.000,C 90.000,E1 127.810} C_DIS
LIN {X 0.192,Y -508.410,Z 395.505,A 0.000,B 0.000,C 90.000,E1 126.870} C_DIS
LIN {X -0.090,Y -507.626,Z 395.500,A 0.000,B 0.000,C 90.000,E1 126.011} C_DIS
LIN {X 0.031,Y -506.416,Z 395.495,A 0.000,B 0.000,C 90.000,E1 125.105} C_DIS
LIN {X 0.034,Y -504.378,Z 395.488,A 0.000,B 0.000,C 90.000,E1 123.913} C_DIS
LIN {X -0.076,Y -503.824,Z 395.487,A 0.000,B 0.000,C 90.000,E1 123.627} C_DIS
LIN {X -0.159,Y -502.379,Z 395.483,A 0.000,B 0.000,C 90.000,E1 123.038} C_DIS
LIN {X 0.193,Y -498.858,Z 395.477,A 0.000,B 0.000,C 90.000,E1 121.799} C_DIS
LIN {X -0.202,Y -497.967,Z 395.475,A 0.000,B 0.000,C 90.000,E1 121.544} C_DIS
LIN {X 0.220,Y -494.778,Z 395.470,A 0.000,B 0.000,C 90.000,E1 120.590} C_DIS
LIN {X -0.062,Y -490.155,Z 395.463,A 0.000,B 0.000,C 90.000,E1 119.411} C_DIS
LIN {X 0.222,Y -486.928,Z 395.459,A 0.000,B 0.000,C 90.000,E1 118.615} C_DIS
LIN {X 0.241,Y -481.475,Z 395.452,A 0.000,B 0.000,C 90.000,E1 117.385} C_DIS
LIN {X -0.053,Y -474.868,Z 395.445,A 0.000,B 0.000,C 90.000,E1 116.027} C_DIS
LIN {X 0.278,Y -471.092,Z 395.440,A 0.000,B 0.000,C 90.000,E1 115.207} C_DIS
LIN {X 0.028,Y -464.072,Z 395.432,A 0.000,B 0.000,C 90.000,E1 113.823} C_DIS
LIN {X -0.010,Y -458.631,Z 395.426,A 0.000,B 0.000,C 90.000,E1 112.717} C_DIS
LIN {X 0.105,Y -452.687,Z 395.419,A 0.000,B 0.000,C 90.000,E1 111.482} C_DIS
LIN {X 0.066,Y -452.693,Z 395.419,A 0.000,B 0.000,C 90.000,E1 111.482} C_DIS
LIN {X -0.044,Y -456.759,Z 395.411,A 0.000,B 0.000,C 90.000,E1 109.993} C_DIS
LIN {X -0.144,Y -457.528,Z 395.409,A 0.000,B 0.000,C 90.000,E1 109.685} C_DIS
LIN {X -0.074,Y -466.213,Z 395.386,A 0.000,B 0.000,C 90.000,E1 105.536} C_DIS
LIN {X -0.022,Y -467.777,Z 395.383,A 0.000,B 0.000,C 90.000,E1 104.898} C_DIS
LIN {X -0.051,Y -475.982,Z 395.357,A 0.000,B 0.000,C 90.000,E1 100.197} C_DIS
LIN {X 0.099,Y -476.686,Z 395.353,A 0.000,B 0.000,C 90.000,E1 99.557} C_DIS
LIN {X 0.224,Y -481.926,Z 395.331,A 0.000,B 0.000,C 90.000,E1 95.511} C_DIS
LIN {X 0.071,Y -482.206,Z 395.329,A 0.000,B 0.000,C 90.000,E1 95.220} C_DIS
LIN {X 0.010,Y -485.398,Z 395.305,A 0.000,B 0.000,C 90.000,E1 90.917} C_DIS
LIN {X -0.167,Y -485.529,Z 395.303,A 0.000,B 0.000,C 90.000,E1 90.630} C_DIS
LIN {X 0.042,Y -486.362,Z 395.281,A 0.000,B 0.000,C 90.000,E1 86.617} C_DIS
LIN {X -0.133,Y -486.368,Z 395.280,A 0.000,B 0.000,C 90.000,E1 86.331} C_DIS
LIN {X -0.144,Y -485.853,Z 395.274,A 0.000,B 0.000,C 90.000,E1 85.412} C_DIS
LIN {X -0.110,Y -484.692,Z 395.254,A 0.000,B 0.000,C 90.000,E1 81.724} C_DIS
LIN {X -0.241,Y -484.497,Z 395.252,A 0.000,B 0.000,C 90.000,E1 81.432} C_DIS
LIN {X 0.097,Y -480.426,Z 395.227,A 0.000,B 0.000,C 90.000,E1 76.769} C_DIS
LIN {X -0.021,Y -474.200,Z 395.201,A 0.000,B 0.000,C 90.000,E1 72.127} C_DIS
LIN {X -0.088,Y -473.032,Z 395.197,A 0.000,B 0.000,C 90.000,E1 71.511} C_DIS
LIN {X -0.025,Y -471.526,Z 395.193,A 0.000,B 0.000,C 90.000,E1 70.732} C_DIS
LIN {X -0.065,Y -471.540,Z 395.193,A 0.000,B 0.000,C 90.000,E1 70.732} C_DIS
LIN {X 0.046,Y -483.070,Z 395.184,A 0.000,B 0.000,C 90.000,E1 69.156} C_DIS
LIN {X 0.097,Y -492.154,Z 395.177,A 0.000,B 0.000,C 90.000,E1 67.922} C_DIS
LIN {X 0.023,Y -499.806,Z 395.172,A 0.000,B 0.000,C 90.000,E1 66.869} C_DIS
LIN {X 0.169,Y -505.002,Z 395.167,A 0.000,B 0.000,C 90.000,E1 66.102} C_DIS
LIN {X 0.066,Y -507.988,Z 395.165,A 0.000,B 0.000,C 90.000,E1 65.665} C_DIS
LIN {X 0.084,Y -512.636,Z 395.161,A 0.000,B 0.000,C 90.000,E1 64.921} C_DIS
LIN {X 0.239,Y -515.267,Z 395.158,A 0.000,B 0.000,C 90.000,E1 64.460} C_DIS
LIN {X 0.191,Y -517.737,Z 395.156,A 0.000,B 0.000,C 90.000,E1 64.024} C_DIS
LIN {X 0.054,Y -521.409,Z 395.152,A 0.000,B 0.000,C 90.000,E1 63.307} C_DIS
LIN {X -0.286,Y -524.886,Z 395.148,A 0.000,B 0.000,C 90.000,E1 62.615} C_DIS
LIN {X -0.049,Y -526.901,Z 395.145,A 0.000,B 0.000,C 90.000,E1 62.153} C_DIS
LIN {X 0.050,Y -529.217,Z 395.142,A 0.000,B 0.000,C 90.000,E1 61.563} C_DIS
LIN {X -0.090,Y -531.357,Z 395.139,A 0.000,B 0.000,C 90.000,E1 61.001} C_DIS
LIN {X 0.009,Y -534.232,Z 395.134,A 0.000,B 0.000,C 90.000,E1 60.127} C_DIS
